C01817=1103.978,373.015,410.367,-179.779,17.252,151.645
C01818=1103.984,373.262,410.332,-179.776,17.255,151.645
C01819=1103.989,373.509,410.296,-179.773,17.259,151.646
C01820=1103.995,373.757,410.260,-179.770,17.264,151.646
C01821=1104.002,374.004,410.224,-179.768,17.268,151.646
C01822=1104.007,374.251,410.189,-179.765,17.272,151.647
C01823=1104.012,374.499,410.152,-179.762,17.276,151.647
C01824=1104.018,374.745,410.116,-179.760,17.280,151.648
C01825=1104.024,374.993,410.081,-179.757,17.284,151.648
C01826=1104.029,375.240,410.045,-179.754,17.289,151.649
C01827=1104.035,375.487,410.008,-179.751,17.293,151.649
C01828=1104.041,375.735,409.972,-179.748,17.297,151.650
C01829=1104.046,375.982,409.936,-179.746,17.302,151.650
C01830=1104.052,376.229,409.900,-179.743,17.306,151.651
C01831=1104.058,376.476,409.865,-179.740,17.310,151.651
C01832=1104.063,376.724,409.828,-179.737,17.314,151.652
C01833=1104.069,376.971,409.792,-179.735,17.319,151.653
C01834=1104.075,377.218,409.756,-179.732,17.323,151.653
C01835=1104.080,377.466,409.719,-179.728,17.328,151.653
C01836=1104.086,377.713,409.684,-179.727,17.332,151.654
C01837=1104.092,377.960,409.648,-179.724,17.336,151.655
C01838=1104.097,378.208,409.611,-179.721,17.341,151.655
C01839=1104.103,378.454,409.575,-179.718,17.345,151.656
C01840=1104.108,378.702,409.539,-179.716,17.349,151.656
C01841=1104.115,378.949,409.502,-179.713,17.354,151.657
C01842=1104.120,379.195,409.466,-179.710,17.358,151.657
C01843=1104.126,379.443,409.430,-179.707,17.363,151.658
C01844=1104.132,379.690,409.394,-179.704,17.368,151.659
C01845=1104.137,379.938,409.357,-179.702,17.372,151.659
C01846=1104.143,380.185,409.321,-179.699,17.376,151.660
C01847=1104.149,380.432,409.284,-179.696,17.381,151.660
C01848=1104.155,380.680,409.248,-179.694,17.385,151.661
C01849=1104.160,380.927,409.212,-179.691,17.390,151.661
C01850=1104.166,381.174,409.175,-179.689,17.394,151.662
C01851=1104.171,381.422,409.139,-179.686,17.399,151.663
C01852=1104.178,381.669,409.103,-179.683,17.404,151.663
C01853=1104.183,381.915,409.066,-179.680,17.408,151.664
C01854=1104.189,382.162,409.029,-179.678,17.413,151.664
C01855=1104.195,382.410,408.992,-179.674,17.417,151.665
C01856=1104.201,382.657,408.957,-179.673,17.422,151.666
C01857=1104.210,383.071,408.895,-179.668,17.430,151.667
C01858=1104.219,383.485,408.834,-179.663,17.438,151.668
C01859=1104.228,383.899,408.773,-179.659,17.446,151.669
C01860=1104.239,384.314,408.711,-179.655,17.454,151.670
C01861=1104.244,384.561,408.674,-179.652,17.458,151.671
C01862=1104.249,384.808,408.637,-179.649,17.463,151.671
C01863=1104.256,385.055,408.601,-179.647,17.468,151.672
C01864=1104.261,385.302,408.564,-179.644,17.473,151.673
C01865=1104.266,385.549,408.527,-179.641,17.478,151.673
C01866=1104.273,385.796,408.491,-179.639,17.483,151.674
C01867=1104.278,386.043,408.454,-179.636,17.488,151.675
C01868=1104.284,386.291,408.417,-179.634,17.493,151.676
C01869=1104.289,386.537,408.380,-179.631,17.498,151.676
C01870=1104.295,386.785,408.343,-179.629,17.502,151.677
C01871=1104.301,387.032,408.306,-179.626,17.507,151.678
C01872=1104.306,387.279,408.269,-179.624,17.512,151.678
C01873=1104.312,387.526,408.232,-179.621,17.517,151.679
C01874=1104.318,387.773,408.195,-179.619,17.522,151.680
C01875=1104.324,388.020,408.159,-179.616,17.527,151.681
C01876=1104.329,388.267,408.121,-179.613,17.532,151.681
C01877=1104.335,388.514,408.084,-179.611,17.537,151.682
C01878=1104.340,388.762,408.047,-179.609,17.542,151.683
C01879=1104.346,389.009,408.010,-179.606,17.547,151.684
C01880=1104.353,389.256,407.973,-179.603,17.552,151.684
C01881=1104.358,389.503,407.936,-179.601,17.557,151.685
C01882=1104.364,389.750,407.899,-179.598,17.563,151.686
C01883=1104.369,389.996,407.862,-179.596,17.568,151.687
C01884=1104.375,390.244,407.825,-179.593,17.573,151.687
C01885=1104.380,390.491,407.788,-179.591,17.578,151.688
C01886=1104.386,390.738,407.750,-179.588,17.583,151.689
C01887=1104.393,390.985,407.713,-179.586,17.588,151.690
C01888=1104.398,391.232,407.676,-179.583,17.593,151.690
C01889=1104.404,391.479,407.639,-179.581,17.599,151.691
C01890=1104.410,391.726,407.602,-179.578,17.604,151.692
C01891=1104.415,391.974,407.565,-179.576,17.609,151.693
C01892=1104.421,392.220,407.527,-179.573,17.615,151.694
C01893=1104.427,392.468,407.490,-179.570,17.620,151.695
C01894=1104.433,392.715,407.452,-179.568,17.625,151.695
C01895=1104.438,392.962,407.415,-179.565,17.631,151.696
C01896=1104.444,393.209,407.377,-179.563,17.636,151.697
C01897=1104.450,393.456,407.340,-179.561,17.641,151.698
C01898=1104.456,393.703,407.302,-179.558,17.646,151.699
C01899=1104.461,393.950,407.265,-179.556,17.652,151.700
C01900=1104.467,394.197,407.228,-179.553,17.657,151.701
C01901=1104.473,394.444,407.191,-179.551,17.663,151.702
C01902=1104.479,394.691,407.153,-179.549,17.668,151.703
C01903=1104.483,394.939,407.115,-179.547,17.673,151.703
C01904=1104.489,395.185,407.077,-179.544,17.679,151.704
C01905=1104.495,395.432,407.040,-179.541,17.685,151.705
C01906=1104.501,395.680,407.003,-179.539,17.690,151.706
C01907=1104.507,395.926,406.965,-179.537,17.696,151.707
C01908=1104.513,396.173,406.927,-179.534,17.701,151.708
C01909=1104.518,396.387,406.895,-179.533,17.706,151.709
C01910=1104.523,396.600,406.862,-179.530,17.711,151.709
C01911=1104.528,396.813,406.830,-179.529,17.716,151.710
C01912=1104.533,397.026,406.797,-179.526,17.721,151.711
C01913=1104.537,397.239,406.764,-179.524,17.725,151.712
C01914=1104.542,397.453,406.731,-179.522,17.731,151.713
C01915=1104.547,397.666,406.699,-179.520,17.735,151.714
C01916=1104.552,397.879,406.666,-179.518,17.741,151.714
C01917=1104.557,398.126,406.629,-179.516,17.746,151.715
C01918=1104.563,398.373,406.592,-179.513,17.752,151.716
C01919=1104.569,398.621,406.553,-179.511,17.757,151.717
C01920=1104.575,398.868,406.515,-179.509,17.763,151.718
C01921=1104.581,399.114,406.477,-179.506,17.769,151.719
C01922=1104.586,399.361,406.440,-179.504,17.775,151.720
C01923=1104.592,399.608,406.401,-179.502,17.781,151.721
C01924=1104.597,399.855,406.364,-179.500,17.786,151.722
C01925=1104.604,400.103,406.326,-179.497,17.793,151.723
C01926=1104.609,400.350,406.288,-179.495,17.798,151.724
C01927=1104.615,400.597,406.250,-179.493,17.804,151.725
C01928=1104.620,400.844,406.212,-179.491,17.810,151.727
C01929=1104.626,401.090,406.174,-179.488,17.816,151.728
C01930=1104.631,401.338,406.136,-179.486,17.822,151.729
C01931=1104.638,401.585,406.098,-179.484,17.828,151.730
C01932=1104.643,401.832,406.060,-179.482,17.834,151.731
C01933=1104.649,402.079,406.021,-179.479,17.840,151.732
C01934=1104.655,402.326,405.984,-179.477,17.846,151.733
C01935=1104.660,402.573,405.945,-179.475,17.852,151.734
C01936=1104.666,402.820,405.907,-179.472,17.859,151.735
C01937=1104.671,403.067,405.869,-179.470,17.865,151.736
C01938=1104.678,403.313,405.830,-179.468,17.871,151.737
C01939=1104.683,403.560,405.792,-179.465,17.877,151.738
C01940=1104.689,403.808,405.754,-179.463,17.883,151.739
C01941=1104.694,404.055,405.716,-179.462,17.889,151.741
C01942=1104.700,404.302,405.678,-179.459,17.896,151.742
C01943=1104.706,404.549,405.639,-179.457,17.902,151.743
C01944=1104.712,404.796,405.600,-179.455,17.908,151.744
C01945=1104.717,405.042,405.562,-179.453,17.915,151.745
C01946=1104.723,405.290,405.524,-179.451,17.921,151.746
C01947=1104.729,405.537,405.486,-179.448,17.928,151.748
C01948=1104.735,405.783,405.447,-179.446,17.933,151.749
C01949=1104.740,406.030,405.408,-179.444,17.940,151.750
C01950=1104.746,406.277,405.371,-179.442,17.946,151.751
C01951=1104.752,406.524,405.331,-179.440,17.953,151.752
C01952=1104.757,406.771,405.293,-179.437,17.960,151.754
C01953=1104.763,407.018,405.255,-179.435,17.965,151.755
C01954=1104.769,407.265,405.216,-179.433,17.972,151.756
C01955=1104.774,407.512,405.177,-179.431,17.979,151.757
C01956=1104.780,407.758,405.139,-179.429,17.986,151.758
C01957=1104.786,408.006,405.100,-179.427,17.992,151.760
C01958=1104.791,408.253,405.062,-179.424,17.999,151.761
C01959=1104.797,408.500,405.023,-179.423,18.005,151.762
C01960=1104.802,408.747,404.984,-179.420,18.012,151.763
C01961=1104.809,408.994,404.945,-179.418,18.018,151.765
C01962=1104.814,409.241,404.907,-179.416,18.026,151.766
C01963=1104.820,409.488,404.868,-179.414,18.032,151.767
C01964=1104.825,409.735,404.829,-179.412,18.039,151.769
C01965=1104.830,409.948,404.795,-179.410,18.045,151.770
C01966=1104.835,410.161,404.762,-179.408,18.051,151.771
C01967=1104.840,410.374,404.728,-179.407,18.056,151.772
C01968=1104.845,410.587,404.696,-179.405,18.062,151.773
C01969=1104.849,410.800,404.662,-179.403,18.068,151.774
C01970=1104.854,411.013,404.628,-179.401,18.074,151.775
C01971=1104.860,411.226,404.595,-179.399,18.080,151.776
C01972=1104.864,411.439,404.561,-179.398,18.086,151.778
C01973=1104.869,411.686,404.522,-179.395,18.093,151.779
C01974=1104.876,411.933,404.483,-179.393,18.100,151.780
C01975=1104.882,412.179,404.444,-179.392,18.107,151.782
C01976=1104.888,412.426,404.405,-179.389,18.114,151.783
C01977=1104.893,412.673,404.367,-179.387,18.121,151.784
C01978=1104.899,412.921,404.327,-179.385,18.128,151.786
C01979=1104.905,413.167,404.288,-179.383,18.135,151.787
C01980=1104.911,413.414,404.249,-179.381,18.142,151.789
C01981=1104.916,413.661,404.210,-179.379,18.149,151.790
C01982=1104.922,413.908,404.171,-179.377,18.156,151.791
C01983=1104.927,414.155,404.132,-179.375,18.164,151.793
C01984=1104.933,414.402,404.092,-179.374,18.171,151.794
C01985=1104.939,414.648,404.053,-179.371,18.178,151.796
C01986=1104.945,414.896,404.014,-179.369,18.185,151.797
C01987=1104.950,415.142,403.975,-179.367,18.193,151.799
C01988=1104.956,415.389,403.935,-179.365,18.200,151.800
C01989=1104.962,415.636,403.896,-179.363,18.207,151.802
C01990=1104.968,415.883,403.857,-179.361,18.215,151.803
C01991=1104.973,416.129,403.818,-179.359,18.222,151.804
C01992=1104.980,416.376,403.778,-179.358,18.229,151.806
C01993=1104.985,416.623,403.739,-179.355,18.236,151.807
C01994=1104.991,416.870,403.700,-179.353,18.244,151.809
C01995=1104.996,417.117,403.660,-179.351,18.252,151.810
C01996=1105.002,417.364,403.621,-179.349,18.259,151.812
C01997=1105.007,417.610,403.582,-179.348,18.267,151.814
C01998=1105.014,417.857,403.542,-179.346,18.274,151.815
C01999=1105.019,418.103,403.502,-179.344,18.282,151.817
C02000=1105.025,418.351,403.462,-179.342,18.290,151.818
C02001=1105.031,418.598,403.423,-179.340,18.297,151.820
C02002=1105.036,418.844,403.384,-179.338,18.305,151.821
C02003=1105.042,419.091,403.344,-179.336,18.313,151.823
C02004=1105.047,419.337,403.304,-179.334,18.321,151.825
C02005=1105.053,419.584,403.265,-179.333,18.328,151.826
C02006=1105.059,419.831,403.226,-179.331,18.336,151.828
C02007=1105.065,420.077,403.185,-179.329,18.344,151.830
C02008=1105.071,420.325,403.145,-179.327,18.352,151.831
C02009=1105.076,420.571,403.106,-179.325,18.360,151.833
C02010=1105.082,420.818,403.066,-179.323,18.368,151.834
C02011=1105.087,421.065,403.027,-179.321,18.375,151.836
C02012=1105.093,421.312,402.987,-179.319,18.383,151.838
C02013=1105.100,421.558,402.947,-179.318,18.392,151.839
C02014=1105.104,421.805,402.907,-179.316,18.400,151.841
C02015=1105.111,422.051,402.867,-179.314,18.408,151.843
C02016=1105.117,422.299,402.828,-179.312,18.416,151.844
C02017=1105.122,422.545,402.787,-179.310,18.424,151.846
C02018=1105.128,422.792,402.748,-179.308,18.432,151.848
C02019=1105.134,423.038,402.708,-179.307,18.440,151.850
C02020=1105.139,423.285,402.668,-179.305,18.448,151.851
C02021=1105.144,423.505,402.632,-179.304,18.455,151.853
C02022=1105.150,423.724,402.597,-179.302,18.463,151.854
C02023=1105.155,423.944,402.561,-179.300,18.470,151.856
C02024=1105.160,424.164,402.526,-179.299,18.477,151.858
C02025=1105.164,424.383,402.490,-179.297,18.485,151.859
C02026=1105.169,424.604,402.454,-179.296,18.492,151.861
C02027=1105.174,424.822,402.418,-179.294,18.500,151.862
C02028=1105.179,425.043,402.382,-179.293,18.507,151.864
C02029=1105.186,425.289,402.342,-179.291,18.516,151.866
C02030=1105.191,425.536,402.303,-179.290,18.524,151.868
C02031=1105.197,425.782,402.262,-179.288,18.533,151.869
C02032=1105.203,426.029,402.222,-179.286,18.542,151.871
C02033=1105.208,426.275,402.182,-179.284,18.550,151.873
C02034=1105.214,426.523,402.142,-179.282,18.559,151.875
C02035=1105.220,426.769,402.102,-179.281,18.567,151.877
C02036=1105.226,427.016,402.061,-179.279,18.576,151.879
C02037=1105.231,427.262,402.021,-179.278,18.584,151.881
C02038=1105.237,427.509,401.980,-179.277,18.593,151.883
C02039=1105.243,427.755,401.940,-179.274,18.602,151.885
C02040=1105.249,428.002,401.900,-179.273,18.611,151.886
C02041=1105.254,428.249,401.860,-179.271,18.619,151.888
C02042=1105.260,428.495,401.819,-179.270,18.628,151.890
C02043=1105.266,428.742,401.779,-179.268,18.637,151.892
C02044=1105.272,428.989,401.738,-179.266,18.646,151.894
C02045=1105.277,429.236,401.698,-179.265,18.655,151.896
C02046=1105.283,429.481,401.658,-179.263,18.664,151.898
C02047=1105.289,429.728,401.617,-179.262,18.673,151.900
C02048=1105.294,429.975,401.576,-179.260,18.682,151.902
C02049=1105.300,430.221,401.535,-179.259,18.691,151.904
C02050=1105.306,430.467,401.495,-179.257,18.700,151.906
C02051=1105.312,430.714,401.454,-179.255,18.710,151.908
C02052=1105.317,430.961,401.414,-179.254,18.719,151.910
C02053=1105.323,431.208,401.373,-179.253,18.728,151.912
C02054=1105.329,431.454,401.332,-179.251,18.737,151.914
C02055=1105.334,431.700,401.292,-179.249,18.747,151.917
C02056=1105.340,431.946,401.251,-179.248,18.756,151.919
C02057=1105.346,432.193,401.210,-179.247,18.765,151.921
C02058=1105.352,432.440,401.169,-179.245,18.775,151.923
C02059=1105.357,432.687,401.129,-179.244,18.784,151.925
C02060=1105.363,432.933,401.087,-179.243,18.793,151.927
C02061=1105.368,433.179,401.047,-179.241,18.803,151.929
C02062=1105.375,433.426,401.007,-179.240,18.812,151.931
C02063=1105.381,433.672,400.965,-179.238,18.822,151.934
C02064=1105.386,433.919,400.924,-179.237,18.832,151.936
C02065=1105.392,434.166,400.884,-179.236,18.841,151.938
C02066=1105.398,434.412,400.842,-179.234,18.851,151.940
C02067=1105.403,434.659,400.802,-179.233,18.861,151.943
C02068=1105.408,434.904,400.760,-179.231,18.870,151.945
C02069=1105.414,435.151,400.719,-179.230,18.880,151.947
C02070=1105.419,435.398,400.678,-179.229,18.890,151.949
C02071=1105.425,435.644,400.637,-179.228,18.900,151.951
C02072=1105.431,435.891,400.596,-179.226,18.910,151.954
C02073=1105.437,436.137,400.555,-179.225,18.919,151.956
C02074=1105.443,436.384,400.513,-179.224,18.930,151.958
C02075=1105.448,436.630,400.472,-179.223,18.940,151.961
C02076=1105.454,436.877,400.431,-179.221,18.950,151.963
C02077=1105.459,437.090,400.395,-179.220,18.958,151.965
C02078=1105.464,437.303,400.360,-179.219,18.967,151.967
C02079=1105.468,437.516,400.324,-179.219,18.976,151.969
C02080=1105.474,437.731,400.288,-179.217,18.985,151.971
C02081=1105.479,437.944,400.253,-179.216,18.994,151.973
C02082=1105.484,438.157,400.216,-179.215,19.002,151.975
C02083=1105.489,438.371,400.181,-179.214,19.011,151.977
C02084=1105.494,438.584,400.145,-179.213,19.020,151.979
C02085=1105.500,438.831,400.104,-179.212,19.030,151.982
C02086=1105.506,439.077,400.063,-179.210,19.041,151.984
C02087=1105.511,439.324,400.021,-179.209,19.052,151.987
C02088=1105.517,439.570,399.980,-179.208,19.062,151.989
C02089=1105.523,439.816,399.938,-179.207,19.072,151.992
C02090=1105.529,440.062,399.897,-179.206,19.083,151.994
C02091=1105.535,440.309,399.855,-179.205,19.093,151.997
C02092=1105.539,440.556,399.814,-179.204,19.104,151.999
C02093=1105.545,440.802,399.772,-179.203,19.114,152.002
C02094=1105.551,441.048,399.731,-179.202,19.125,152.004
C02095=1105.557,441.294,399.689,-179.200,19.136,152.007
C02096=1105.562,441.541,399.647,-179.200,19.147,152.009
C02097=1105.568,441.787,399.606,-179.199,19.158,152.012
C02098=1105.574,442.033,399.564,-179.197,19.169,152.014
C02099=1105.580,442.280,399.522,-179.197,19.179,152.017
C02100=1105.586,442.526,399.481,-179.196,19.190,152.020
C02101=1105.591,442.772,399.439,-179.195,19.202,152.022
C02102=1105.597,443.018,399.397,-179.194,19.212,152.025
C02103=1105.603,443.264,399.355,-179.193,19.223,152.028
C02104=1105.608,443.511,399.313,-179.192,19.235,152.030
C02105=1105.614,443.757,399.272,-179.191,19.245,152.033
C02106=1105.620,444.004,399.229,-179.190,19.257,152.036
C02107=1105.626,444.250,399.188,-179.190,19.268,152.039
C02108=1105.631,444.497,399.146,-179.190,19.278,152.041
C02109=1105.637,444.743,399.104,-179.190,19.290,152.044
C02110=1105.643,444.989,399.062,-179.190,19.301,152.047
C02111=1105.648,445.235,399.020,-179.190,19.312,152.050
C02112=1105.654,445.482,398.978,-179.190,19.323,152.053
C02113=1105.660,445.727,398.936,-179.190,19.333,152.055
C02114=1105.666,445.975,398.894,-179.190,19.345,152.058
C02115=1105.672,446.221,398.852,-179.191,19.355,152.061
C02116=1105.677,446.467,398.810,-179.192,19.366,152.064
C02117=1105.683,446.713,398.768,-179.192,19.377,152.067
C02118=1105.688,446.959,398.726,-179.193,19.388,152.070
C02119=1105.694,447.206,398.684,-179.194,19.399,152.073
C02120=1105.700,447.452,398.642,-179.195,19.410,152.076
C02121=1105.706,447.699,398.599,-179.197,19.421,152.079
C02122=1105.711,447.945,398.557,-179.198,19.432,152.082
C02123=1105.717,448.191,398.515,-179.199,19.443,152.085
C02124=1105.722,448.437,398.473,-179.201,19.453,152.088
C02125=1105.728,448.683,398.430,-179.201,19.464,152.091
C02126=1105.734,448.930,398.388,-179.203,19.475,152.094
C02127=1105.740,449.177,398.346,-179.205,19.486,152.097
C02128=1105.745,449.423,398.303,-179.207,19.496,152.100
C02129=1105.751,449.669,398.262,-179.209,19.507,152.103
C02130=1105.757,449.915,398.219,-179.211,19.517,152.106
C02131=1105.762,450.162,398.177,-179.213,19.529,152.109
C02132=1105.769,450.407,398.135,-179.215,19.539,152.112
C02133=1105.364,450.401,398.011,-179.292,19.769,152.185
C02134=1105.357,450.155,398.053,-179.290,19.758,152.182
C02135=1105.352,449.909,398.095,-179.288,19.747,152.179
C02136=1105.346,449.662,398.138,-179.286,19.736,152.175
C02137=1105.340,449.416,398.180,-179.284,19.726,152.172
C02138=1105.335,449.170,398.222,-179.283,19.715,152.169
C02139=1105.329,448.924,398.265,-179.282,19.704,152.166
C02140=1105.323,448.678,398.307,-179.280,19.693,152.163
C02141=1105.317,448.431,398.349,-179.278,19.682,152.160
C02142=1105.312,448.185,398.392,-179.277,19.671,152.157
C02143=1105.307,447.938,398.434,-179.275,19.661,152.154
C02144=1105.301,447.692,398.475,-179.274,19.649,152.151
C02145=1105.294,447.446,398.519,-179.273,19.638,152.148
C02146=1105.289,447.199,398.561,-179.273,19.627,152.145
C02147=1105.283,446.953,398.603,-179.272,19.616,152.142
C02148=1105.278,446.707,398.645,-179.271,19.605,152.139
C02149=1105.273,446.460,398.687,-179.270,19.594,152.136
C02150=1105.266,446.215,398.729,-179.269,19.583,152.133
C02151=1105.260,445.968,398.771,-179.269,19.572,152.130
C02152=1105.255,445.721,398.813,-179.268,19.561,152.127
C02153=1105.249,445.476,398.856,-179.269,19.550,152.125
C02154=1105.243,445.229,398.897,-179.268,19.539,152.122
C02155=1105.238,444.983,398.939,-179.268,19.528,152.119
C02156=1105.231,444.737,398.982,-179.268,19.517,152.116
C02157=1105.226,444.490,399.024,-179.268,19.506,152.113
C02158=1105.220,444.244,399.065,-179.269,19.495,152.111
C02159=1105.215,443.997,399.107,-179.270,19.483,152.108
C02160=1105.208,443.752,399.149,-179.270,19.473,152.105
C02161=1105.203,443.505,399.192,-179.271,19.461,152.102
C02162=1105.197,443.259,399.233,-179.272,19.450,152.100
C02163=1105.192,443.013,399.275,-179.273,19.439,152.097
C02164=1105.186,442.766,399.316,-179.274,19.428,152.094
C02165=1105.181,442.520,399.359,-179.274,19.417,152.092
C02166=1105.174,442.274,399.401,-179.276,19.406,152.089
C02167=1105.168,442.027,399.443,-179.277,19.395,152.086
C02168=1105.163,441.781,399.485,-179.278,19.383,152.084
C02169=1105.157,441.535,399.526,-179.279,19.373,152.081
C02170=1105.151,441.288,399.567,-179.280,19.362,152.079
C02171=1105.146,441.042,399.610,-179.281,19.351,152.076
C02172=1105.140,440.796,399.651,-179.282,19.340,152.074
C02173=1105.134,440.549,399.692,-179.283,19.329,152.071
C02174=1105.129,440.303,399.735,-179.285,19.319,152.068
C02175=1105.123,440.057,399.776,-179.286,19.309,152.066
C02176=1105.117,439.811,399.817,-179.287,19.298,152.064
C02177=1105.111,439.564,399.859,-179.288,19.287,152.061
C02178=1105.105,439.318,399.900,-179.289,19.277,152.059
C02179=1105.100,439.071,399.942,-179.291,19.266,152.056
C02180=1105.094,438.825,399.983,-179.291,19.256,152.054
C02181=1105.088,438.579,400.025,-179.293,19.245,152.051
C02182=1105.083,438.367,400.060,-179.294,19.236,152.049
C02183=1105.078,438.156,400.096,-179.295,19.228,152.047
C02184=1105.073,437.945,400.131,-179.296,19.218,152.045
C02185=1105.068,437.733,400.167,-179.297,19.210,152.043
C02186=1105.063,437.522,400.202,-179.298,19.201,152.041
C02187=1105.058,437.311,400.237,-179.300,19.192,152.039
C02188=1105.054,437.100,400.272,-179.300,19.184,152.037
C02189=1105.048,436.889,400.309,-179.302,19.175,152.035
C02190=1105.042,436.642,400.349,-179.303,19.165,152.033
C02191=1105.037,436.396,400.390,-179.304,19.154,152.030
C02192=1105.031,436.149,400.431,-179.305,19.145,152.028
C02193=1105.025,435.903,400.473,-179.307,19.134,152.026
C02194=1105.017,435.527,400.536,-179.309,19.119,152.022
C02195=1105.008,435.152,400.598,-179.311,19.104,152.019
C02196=1104.999,434.776,400.662,-179.313,19.089,152.015
C02197=1104.991,434.401,400.724,-179.315,19.074,152.012
C02198=1104.985,434.154,400.765,-179.317,19.064,152.009
C02199=1104.979,433.908,400.805,-179.318,19.055,152.007
C02200=1104.974,433.662,400.846,-179.320,19.045,152.005
C02201=1104.968,433.415,400.887,-179.321,19.035,152.003
C02202=1104.962,433.169,400.929,-179.322,19.026,152.001
C02203=1104.957,432.922,400.969,-179.324,19.016,151.999
C02204=1104.951,432.675,401.010,-179.325,19.007,151.996
C02205=1104.944,432.430,401.051,-179.327,18.997,151.994
C02206=1104.939,432.183,401.092,-179.328,18.988,151.992
C02207=1104.933,431.936,401.133,-179.329,18.978,151.990
C02208=1104.928,431.690,401.173,-179.332,18.969,151.988
C02209=1104.922,431.444,401.214,-179.333,18.959,151.986
C02210=1104.917,431.197,401.255,-179.334,18.950,151.984
C02211=1104.911,430.950,401.296,-179.336,18.941,151.982
C02212=1104.905,430.703,401.336,-179.337,18.932,151.980
C02213=1104.899,430.457,401.376,-179.339,18.922,151.978
C02214=1104.894,430.211,401.418,-179.340,18.914,151.976
C02215=1104.888,429.964,401.459,-179.342,18.904,151.973
C02216=1104.882,429.717,401.499,-179.344,18.895,151.971
C02217=1104.876,429.471,401.539,-179.345,18.886,151.970
C02218=1104.871,429.225,401.580,-179.347,18.876,151.967
C02219=1104.865,428.978,401.621,-179.348,18.868,151.965
C02220=1104.859,428.731,401.661,-179.350,18.859,151.963
C02221=1104.853,428.485,401.701,-179.351,18.850,151.961
C02222=1104.848,428.238,401.742,-179.353,18.841,151.960
C02223=1104.841,427.991,401.782,-179.355,18.832,151.958
C02224=1104.836,427.745,401.823,-179.357,18.823,151.956
C02225=1104.830,427.498,401.863,-179.358,18.814,151.954
C02226=1104.824,427.252,401.904,-179.360,18.806,151.952
C02227=1104.818,427.005,401.944,-179.361,18.797,151.950
C02228=1104.813,426.759,401.984,-179.364,18.788,151.948
C02229=1104.807,426.512,402.024,-179.365,18.779,151.946
C02230=1104.802,426.265,402.065,-179.367,18.771,151.944
C02231=1104.795,426.018,402.105,-179.368,18.762,151.942
C02232=1104.790,425.772,402.145,-179.370,18.754,151.941
C02233=1104.784,425.526,402.186,-179.372,18.745,151.939
C02234=1104.779,425.278,402.226,-179.374,18.736,151.937
C02235=1104.773,425.031,402.266,-179.376,18.728,151.935
C02236=1104.767,424.786,402.306,-179.377,18.719,151.933
C02237=1104.761,424.539,402.347,-179.379,18.711,151.931
C02238=1104.754,424.228,402.397,-179.381,18.700,151.929
C02239=1104.747,423.917,402.447,-179.383,18.690,151.927
C02240=1104.740,423.607,402.498,-179.386,18.679,151.925
C02241=1104.733,423.296,402.548,-179.387,18.669,151.922
C02242=1104.727,423.050,402.588,-179.389,18.661,151.921
C02243=1104.721,422.802,402.628,-179.392,18.652,151.919
C02244=1104.715,422.556,402.668,-179.393,18.644,151.917
C02245=1104.710,422.309,402.708,-179.395,18.636,151.915
C02246=1104.704,422.063,402.748,-179.397,18.627,151.914
C02247=1104.698,421.816,402.788,-179.399,18.619,151.912
C02248=1104.693,421.569,402.828,-179.401,18.611,151.910
C02249=1104.687,421.322,402.867,-179.403,18.603,151.909
C02250=1104.680,421.076,402.908,-179.404,18.596,151.907
C02251=1104.676,420.829,402.947,-179.406,18.588,151.905
C02252=1104.670,420.582,402.987,-179.408,18.580,151.904
C02253=1104.664,420.336,403.026,-179.410,18.572,151.902
C02254=1104.658,420.089,403.066,-179.411,18.564,151.900
C02255=1104.652,419.842,403.107,-179.414,18.556,151.899
C02256=1104.647,419.596,403.146,-179.415,18.548,151.897
C02257=1104.641,419.349,403.185,-179.417,18.540,151.895
C02258=1104.636,419.102,403.225,-179.419,18.532,151.894
C02259=1104.629,418.855,403.265,-179.421,18.524,151.892
C02260=1104.623,418.608,403.304,-179.423,18.517,151.891
C02261=1104.618,418.362,403.343,-179.425,18.508,151.889
C02262=1104.613,418.114,403.383,-179.427,18.501,151.887
C02263=1104.607,417.869,403.423,-179.429,18.494,151.886
C02264=1104.601,417.621,403.463,-179.431,18.486,151.884
C02265=1104.595,417.375,403.502,-179.433,18.478,151.883
C02266=1104.589,417.128,403.541,-179.435,18.470,151.881
C02267=1104.584,416.881,403.581,-179.437,18.463,151.880
C02268=1104.578,416.634,403.620,-179.439,18.455,151.878
C02269=1104.572,416.387,403.660,-179.440,18.448,151.877
C02270=1104.567,416.140,403.699,-179.443,18.441,151.875
C02271=1104.561,415.893,403.738,-179.445,18.433,151.874
C02272=1104.555,415.647,403.778,-179.447,18.425,151.872
C02273=1104.549,415.400,403.817,-179.448,18.419,151.871
C02274=1104.543,415.154,403.856,-179.451,18.411,151.869
C02275=1104.537,414.907,403.896,-179.453,18.404,151.868
C02276=1104.532,414.660,403.934,-179.455,18.396,151.866
C02277=1104.526,414.412,403.974,-179.457,18.389,151.865
C02278=1104.521,414.166,404.013,-179.459,18.382,151.863
C02279=1104.515,413.919,404.052,-179.461,18.374,151.862
C02280=1104.509,413.672,404.091,-179.463,18.367,151.861
C02281=1104.503,413.425,404.131,-179.465,18.360,151.859
C02282=1104.498,413.179,404.170,-179.467,18.353,151.858
C02283=1104.491,412.932,404.209,-179.469,18.345,151.856
C02284=1104.486,412.685,404.247,-179.471,18.339,151.855
C02285=1104.480,412.438,404.287,-179.473,18.331,151.854
C02286=1104.475,412.191,404.326,-179.476,18.324,151.852
C02287=1104.469,411.944,404.365,-179.477,18.318,151.851
C02288=1104.463,411.698,404.404,-179.479,18.310,151.849
C02289=1104.457,411.450,404.443,-179.482,18.303,151.848
C02290=1104.452,411.237,404.477,-179.483,18.298,151.847
C02291=1104.447,411.024,404.510,-179.485,18.291,151.846
C02292=1104.442,410.811,404.544,-179.487,18.285,151.845
C02293=1104.437,410.597,404.577,-179.489,18.279,151.843
C02294=1104.433,410.384,404.611,-179.491,18.273,151.842
C02295=1104.428,410.171,404.645,-179.493,18.267,151.841
C02296=1104.423,409.957,404.678,-179.495,18.261,151.840
C02297=1104.418,409.744,404.712,-179.496,18.256,151.839
C02298=1104.412,409.498,404.751,-179.498,18.249,151.838
C02299=1104.407,409.250,404.789,-179.500,18.242,151.836
C02300=1104.401,409.004,404.828,-179.502,18.235,151.835
C02301=1104.396,408.757,404.867,-179.505,18.228,151.834
C02302=1104.389,408.510,404.906,-179.507,18.222,151.832
C02303=1104.384,408.263,404.944,-179.509,18.215,151.831
C02304=1104.379,408.016,404.983,-179.511,18.208,151.830
C02305=1104.373,407.769,405.022,-179.513,18.201,151.829
C02306=1104.367,407.522,405.060,-179.515,18.195,151.827
C02307=1104.361,407.275,405.099,-179.518,18.188,151.826
C02308=1104.355,407.028,405.138,-179.520,18.182,151.825
C02309=1104.350,406.781,405.176,-179.522,18.175,151.824
C02310=1104.344,406.534,405.214,-179.524,18.169,151.822
C02311=1104.338,406.287,405.254,-179.527,18.162,151.821
C02312=1104.333,406.040,405.292,-179.528,18.155,151.820
C02313=1104.327,405.794,405.330,-179.530,18.150,151.819
C02314=1104.321,405.546,405.369,-179.533,18.143,151.818
C02315=1104.316,405.299,405.407,-179.535,18.136,151.816
C02316=1104.310,405.053,405.445,-179.538,18.130,151.815
C02317=1104.304,404.805,405.485,-179.539,18.123,151.814
C02318=1104.298,404.559,405.522,-179.542,18.117,151.813
C02319=1104.293,404.312,405.561,-179.544,18.111,151.812
C02320=1104.287,404.065,405.599,-179.546,18.105,151.811
C02321=1104.281,403.817,405.637,-179.549,18.098,151.810
C02322=1104.276,403.571,405.676,-179.551,18.092,151.808
C02323=1104.270,403.324,405.714,-179.553,18.086,151.807
C02324=1104.264,403.076,405.753,-179.555,18.080,151.806
C02325=1104.258,402.829,405.791,-179.557,18.074,151.805
C02326=1104.253,402.582,405.829,-179.559,18.068,151.804
C02327=1104.247,402.336,405.867,-179.562,18.061,151.803
C02328=1104.242,402.089,405.905,-179.564,18.055,151.802
C02329=1104.235,401.841,405.943,-179.566,18.049,151.801
C02330=1104.230,401.594,405.981,-179.569,18.042,151.799
C02331=1104.224,401.347,406.019,-179.571,18.037,151.798
C02332=1104.218,401.101,406.057,-179.573,18.031,151.797
C02333=1104.213,400.854,406.095,-179.576,18.025,151.796
C02334=1104.207,400.606,406.133,-179.578,18.019,151.795
C02335=1104.202,400.359,406.172,-179.580,18.013,151.794
C02336=1104.196,400.112,406.210,-179.582,18.007,151.793
C02337=1104.190,399.866,406.247,-179.585,18.000,151.792
C02338=1104.185,399.619,406.286,-179.587,17.995,151.791
C02339=1104.178,399.371,406.324,-179.589,17.989,151.790
C02340=1104.172,399.124,406.362,-179.591,17.983,151.789
C02341=1104.167,398.877,406.400,-179.594,17.977,151.788
C02342=1104.161,398.631,406.438,-179.597,17.971,151.787
C02343=1104.155,398.384,406.475,-179.599,17.965,151.786
C02344=1104.150,398.136,406.513,-179.601,17.960,151.785
C02345=1104.144,397.889,406.551,-179.603,17.954,151.784
C02346=1104.139,397.676,406.583,-179.605,17.949,151.783
C02347=1104.134,397.462,406.616,-179.607,17.944,151.782
C02348=1104.129,397.249,406.649,-179.609,17.939,151.781
C02349=1104.124,397.036,406.681,-179.611,17.934,151.781
C02350=1104.120,396.822,406.714,-179.614,17.929,151.780
C02351=1104.115,396.609,406.747,-179.615,17.924,151.779
C02352=1104.110,396.396,406.780,-179.618,17.919,151.778
C02353=1104.105,396.183,406.812,-179.620,17.915,151.777
C02354=1104.099,395.935,406.850,-179.622,17.909,151.776
C02355=1104.093,395.688,406.887,-179.625,17.903,151.775
C02356=1104.087,395.441,406.925,-179.627,17.897,151.775
C02357=1104.082,395.194,406.963,-179.629,17.892,151.774
C02358=1104.076,394.947,407.000,-179.632,17.886,151.773
C02359=1104.070,394.700,407.038,-179.634,17.881,151.772
C02360=1104.065,394.453,407.075,-179.636,17.875,151.771
C02361=1104.059,394.206,407.113,-179.639,17.870,151.770
C02362=1104.053,393.959,407.150,-179.641,17.865,151.769
C02363=1104.047,393.712,407.187,-179.643,17.859,151.768
C02364=1104.041,393.465,407.225,-179.647,17.853,151.767
C02365=1104.036,393.218,407.262,-179.649,17.848,151.766
C02366=1104.030,392.971,407.300,-179.651,17.842,151.766
C02367=1104.025,392.723,407.338,-179.654,17.837,151.765
C02368=1104.019,392.477,407.375,-179.656,17.832,151.764
C02369=1104.014,392.229,407.412,-179.659,17.827,151.763
C02370=1104.007,391.982,407.449,-179.661,17.821,151.762
C02371=1104.001,391.735,407.487,-179.663,17.816,151.761
C02372=1103.996,391.488,407.524,-179.666,17.811,151.761
C02373=1103.990,391.241,407.561,-179.668,17.806,151.760
C02374=1103.984,390.994,407.598,-179.671,17.801,151.759
C02375=1103.979,390.747,407.636,-179.673,17.795,151.758
C02376=1103.973,390.500,407.673,-179.676,17.790,151.757
C02377=1103.967,390.252,407.710,-179.678,17.785,151.756
C02378=1103.962,390.005,407.747,-179.681,17.780,151.756
C02379=1103.955,389.759,407.785,-179.683,17.774,151.755
C02380=1103.950,389.512,407.821,-179.686,17.769,151.754
C02381=1103.944,389.265,407.858,-179.688,17.764,151.753
C02382=1103.938,389.018,407.896,-179.691,17.759,151.753
C02383=1103.933,388.771,407.933,-179.693,17.754,151.752
C02384=1103.927,388.523,407.970,-179.696,17.749,151.751
C02385=1103.921,388.276,408.007,-179.699,17.743,151.750
C02386=1103.915,388.029,408.044,-179.702,17.738,151.750
C02387=1103.909,387.782,408.081,-179.704,17.734,151.749
C02388=1103.904,387.535,408.118,-179.706,17.729,151.748
C02389=1103.899,387.288,408.155,-179.709,17.723,151.747
C02390=1103.892,387.041,408.191,-179.712,17.719,151.747
C02391=1103.887,386.794,408.229,-179.714,17.714,151.746
C02392=1103.881,386.546,408.266,-179.717,17.708,151.745
C02393=1103.876,386.299,408.303,-179.719,17.704,151.744
C02394=1103.870,386.052,408.339,-179.722,17.699,151.744
C02395=1103.864,385.805,408.376,-179.724,17.693,151.743
C02396=1103.859,385.558,408.413,-179.727,17.689,151.742
C02397=1103.853,385.311,408.450,-179.730,17.684,151.741
C02398=1103.847,385.064,408.487,-179.733,17.679,151.741
C02399=1103.842,384.817,408.523,-179.735,17.674,151.740
C02400=1103.836,384.569,408.560,-179.738,17.669,151.739
C02401=1103.831,384.322,408.597,-179.740,17.664,151.739
C02402=1103.821,383.908,408.658,-179.745,17.656,151.738
C02403=1103.812,383.493,408.720,-179.749,17.648,151.736
C02404=1103.802,383.079,408.782,-179.754,17.640,151.735
C02405=1103.792,382.665,408.843,-179.758,17.632,151.734
C02406=1103.786,382.417,408.880,-179.761,17.627,151.734
C02407=1103.781,382.170,408.915,-179.764,17.622,151.733
C02408=1103.775,381.923,408.952,-179.766,17.618,151.732
C02409=1103.769,381.676,408.989,-179.769,17.613,151.732
C02410=1103.763,381.429,409.026,-179.771,17.609,151.731
C02411=1103.758,381.182,409.061,-179.774,17.604,151.730
C02412=1103.752,380.934,409.098,-179.777,17.599,151.730
C02413=1103.746,380.687,409.135,-179.780,17.594,151.729
C02414=1103.740,380.440,409.172,-179.782,17.590,151.729
C02415=1103.735,380.193,409.207,-179.785,17.586,151.728
C02416=1103.729,379.945,409.244,-179.788,17.581,151.727
C02417=1103.723,379.698,409.281,-179.790,17.576,151.727
C02418=1103.718,379.451,409.316,-179.793,17.572,151.726
C02419=1103.712,379.204,409.353,-179.796,17.567,151.726
C02420=1103.706,378.956,409.389,-179.798,17.563,151.725
C02421=1103.701,378.710,409.425,-179.801,17.559,151.725
C02422=1103.695,378.463,409.462,-179.804,17.554,151.724
C02423=1103.689,378.215,409.498,-179.807,17.549,151.723
C02424=1103.684,377.968,409.534,-179.810,17.545,151.723
C02425=1103.678,377.721,409.570,-179.812,17.541,151.722
C02426=1103.672,377.473,409.607,-179.815,17.536,151.722
C02427=1103.667,377.226,409.642,-179.818,17.532,151.721
C02428=1103.661,376.979,409.680,-179.821,17.527,151.721
C02429=1103.655,376.731,409.715,-179.823,17.523,151.720
C02430=1103.649,376.484,409.751,-179.826,17.519,151.720
C02431=1103.644,376.237,409.788,-179.829,17.514,151.719
C02432=1103.638,375.990,409.823,-179.832,17.510,151.719
C02433=1103.632,375.743,409.859,-179.834,17.505,151.718
C02434=1103.627,375.495,409.896,-179.837,17.501,151.717
C02435=1103.621,375.248,409.931,-179.840,17.497,151.717
C02436=1103.615,375.001,409.968,-179.843,17.493,151.717
C02437=1103.610,374.754,410.004,-179.846,17.488,151.716
C02438=1103.604,374.506,410.039,-179.848,17.484,151.715
C02439=1103.598,374.259,410.076,-179.851,17.480,151.715
C02440=1103.593,374.012,410.111,-179.854,17.475,151.714
C02441=1103.587,373.764,410.147,-179.856,17.472,151.714
C02442=1103.582,373.517,410.183,-179.859,17.467,151.714
C02443=1103.575,373.270,410.219,-179.862,17.463,151.713
C02444=1103.569,373.022,410.255,-179.865,17.459,151.713
C02445=1103.564,372.775,410.290,-179.868,17.455,151.712
C02446=1103.558,372.528,410.326,-179.871,17.451,151.712
C02447=1103.553,372.281,410.361,-179.874,17.446,151.711
C02448=1103.546,372.034,410.398,-179.876,17.443,151.711
C02449=1103.542,371.786,410.434,-179.879,17.439,151.710
C02450=1103.536,371.539,410.470,-179.882,17.434,151.710
C02451=1103.529,371.291,410.505,-179.885,17.430,151.709
C02452=1103.524,371.044,410.541,-179.888,17.426,151.709
C02453=1103.518,370.796,410.576,-179.891,17.422,151.709
C02454=1103.509,370.409,410.632,-179.895,17.416,151.708
C02455=1103.500,370.021,410.688,-179.899,17.410,151.707
C02456=1103.491,369.633,410.744,-179.904,17.404,151.707
C02457=1103.483,369.246,410.799,-179.909,17.397,151.706
C02458=1103.477,368.999,410.835,-179.911,17.393,151.706
C02459=1103.471,368.752,410.871,-179.914,17.389,151.705
C02460=1103.465,368.504,410.906,-179.917,17.385,151.705
C02461=1103.460,368.257,410.941,-179.920,17.381,151.704
C02462=1103.454,368.009,410.977,-179.923,17.377,151.704
C02463=1103.449,367.762,411.012,-179.926,17.373,151.704
C02464=1103.443,367.514,411.048,-179.929,17.370,151.703
C02465=1103.437,367.267,411.083,-179.932,17.365,151.703
C02466=1103.431,367.020,411.119,-179.934,17.362,151.702
C02467=1103.426,366.773,411.154,-179.937,17.358,151.702
C02468=1103.421,366.525,411.189,-179.940,17.354,151.702
C02469=1103.415,366.277,411.225,-179.943,17.350,151.701
C02470=1103.409,366.030,411.260,-179.946,17.346,151.701
C02471=1103.403,365.783,411.296,-179.949,17.343,151.701
C02472=1103.398,365.535,411.330,-179.952,17.339,151.700
C02473=1103.391,365.288,411.365,-179.955,17.335,151.700
C02474=1103.386,365.041,411.401,-179.958,17.331,151.700
C02475=1103.381,364.793,411.435,-179.961,17.327,151.699
C02476=1103.375,364.546,411.471,-179.964,17.324,151.699
C02477=1103.369,364.299,411.507,-179.967,17.320,151.699
C02478=1103.363,364.051,411.541,-179.969,17.316,151.698
C02479=1103.357,363.804,411.576,-179.973,17.312,151.698
C02480=1103.351,363.556,411.612,-179.975,17.309,151.698
C02481=1103.346,363.308,411.647,-179.978,17.305,151.697
C02482=1103.341,363.061,411.682,-179.982,17.301,151.697
C02483=1103.334,362.813,411.717,-179.984,17.298,151.697
C02484=1103.329,362.566,411.752,-179.988,17.294,151.696
C02485=1103.324,362.319,411.787,-179.990,17.291,151.696
C02486=1103.318,362.071,411.822,-179.994,17.287,151.696
C02487=1103.312,361.824,411.856,-179.996,17.283,151.696
C02488=1103.306,361.576,411.892,-180.000,17.280,151.695
C02489=1103.301,361.329,411.927,179.998,17.276,151.695
C02490=1103.295,361.082,411.961,179.995,17.272,151.695
C02491=1103.289,360.834,411.996,179.992,17.269,151.694
C02492=1103.283,360.587,412.032,179.989,17.265,151.694
C02493=1103.278,360.339,412.066,179.986,17.262,151.694
C02494=1103.272,360.091,412.101,179.983,17.258,151.694
C02495=1103.266,359.844,412.136,179.980,17.255,151.693
C02496=1103.261,359.597,412.170,179.977,17.251,151.693
C02497=1103.255,359.349,412.206,179.974,17.248,151.693
C02498=1103.249,359.102,412.241,179.970,17.244,151.693
C02499=1103.244,358.854,412.275,179.968,17.241,151.692
C02500=1103.238,358.606,412.310,179.965,17.237,151.692
C02501=1103.232,358.359,412.345,179.962,17.234,151.692
C02502=1103.227,358.112,412.379,179.958,17.230,151.692
C02503=1103.221,357.864,412.413,179.956,17.227,151.691
C02504=1103.215,357.616,412.448,179.952,17.223,151.691
C02505=1103.209,357.369,412.483,179.949,17.220,151.691
C02506=1103.200,356.996,412.536,179.945,17.215,151.691
C02507=1103.192,356.624,412.587,179.941,17.210,151.690
C02508=1103.183,356.251,412.639,179.936,17.205,151.690
C02509=1103.175,355.878,412.692,179.931,17.200,151.690
C02510=1103.169,355.631,412.726,179.928,17.197,151.689
C02511=1103.163,355.383,412.761,179.925,17.193,151.689
C02512=1103.158,355.135,412.795,179.922,17.190,151.689
C02513=1103.152,354.888,412.829,179.919,17.187,151.689
C02514=1103.147,354.641,412.863,179.916,17.183,151.689
C02515=1103.142,354.393,412.898,179.913,17.180,151.688
C02516=1103.135,354.145,412.933,179.910,17.176,151.688
C02517=1103.129,353.898,412.967,179.907,17.173,151.688
C02518=1103.124,353.650,413.001,179.903,17.170,151.688
C02519=1103.118,353.403,413.035,179.900,17.167,151.688
C02520=1103.113,353.155,413.070,179.898,17.164,151.688
C02521=1103.107,352.907,413.104,179.894,17.160,151.687
C02522=1103.101,352.660,413.138,179.891,17.157,151.687
C02523=1103.096,352.412,413.173,179.888,17.153,151.687
C02524=1103.090,352.165,413.207,179.885,17.151,151.687
C02525=1103.084,351.917,413.240,179.882,17.148,151.687
C02526=1103.078,351.669,413.275,179.879,17.144,151.687
C02527=1103.073,351.422,413.310,179.876,17.141,151.686
C02528=1103.067,351.174,413.344,179.873,17.138,151.686
C02529=1103.061,350.927,413.378,179.869,17.135,151.686
C02530=1103.056,350.679,413.412,179.867,17.132,151.686
C02531=1103.050,350.432,413.446,179.863,17.128,151.686
C02532=1103.044,350.184,413.480,179.860,17.126,151.686
C02533=1103.038,349.936,413.514,179.857,17.123,151.686
C02534=1103.033,349.689,413.549,179.854,17.119,151.685
C02535=1103.027,349.441,413.582,179.851,17.116,151.685
C02536=1103.021,349.194,413.616,179.848,17.113,151.685
C02537=1103.016,348.946,413.650,179.844,17.110,151.685
C02538=1103.011,348.698,413.684,179.841,17.107,151.685
C02539=1103.005,348.451,413.718,179.838,17.104,151.685
C02540=1102.998,348.203,413.753,179.835,17.101,151.685
C02541=1102.993,347.955,413.786,179.832,17.098,151.685
C02542=1102.987,347.708,413.820,179.829,17.095,151.685
C02543=1102.981,347.460,413.854,179.825,17.092,151.684
C02544=1102.976,347.212,413.888,179.823,17.089,151.684
C02545=1102.970,346.965,413.922,179.820,17.086,151.684
C02546=1102.965,346.717,413.955,179.816,17.083,151.684
C02547=1102.959,346.470,413.989,179.813,17.080,151.684
C02548=1102.953,346.222,414.023,179.810,17.077,151.684
C02549=1102.948,345.974,414.057,179.807,17.074,151.684
C02550=1102.942,345.727,414.090,179.804,17.071,151.684
C02551=1102.936,345.479,414.124,179.800,17.068,151.684
C02552=1102.931,345.231,414.158,179.798,17.065,151.684
C02553=1102.925,344.984,414.192,179.794,17.062,151.684
C02554=1102.919,344.736,414.225,179.791,17.059,151.683
C02555=1102.913,344.489,414.259,179.788,17.056,151.683
C02556=1102.908,344.241,414.292,179.785,17.054,151.683
C02557=1102.902,343.992,414.326,179.781,17.050,151.683
C02558=1102.893,343.622,414.377,179.777,17.046,151.683
C02559=1102.885,343.252,414.427,179.772,17.042,151.683
C02560=1102.876,342.882,414.477,179.767,17.038,151.683
C02561=1102.868,342.510,414.528,179.762,17.034,151.683
C02562=1102.862,342.264,414.560,179.760,17.031,151.683
C02563=1102.857,342.016,414.594,179.756,17.028,151.683
C02564=1102.851,341.768,414.627,179.753,17.025,151.683
C02565=1102.845,341.521,414.661,179.750,17.022,151.683
C02566=1102.840,341.273,414.694,179.747,17.020,151.683
C02567=1102.834,341.025,414.728,179.743,17.017,151.683
C02568=1102.828,340.777,414.761,179.740,17.014,151.683
C02569=1102.823,340.529,414.794,179.737,17.011,151.683
C02570=1102.817,340.282,414.828,179.734,17.009,151.683
C02571=1102.812,340.034,414.862,179.730,17.005,151.683
C02572=1102.805,339.786,414.895,179.727,17.003,151.683
C02573=1102.800,339.538,414.928,179.724,17.000,151.683
C02574=1102.794,339.290,414.961,179.721,16.997,151.683
C02575=1102.789,339.042,414.995,179.718,16.995,151.683
C02576=1102.783,338.794,415.028,179.714,16.992,151.683
C02577=1102.777,338.547,415.061,179.711,16.989,151.683
C02578=1102.771,338.299,415.094,179.708,16.987,151.683
C02579=1102.766,338.052,415.127,179.705,16.984,151.683
C02580=1102.761,337.804,415.160,179.702,16.982,151.683
C02581=1102.754,337.556,415.193,179.698,16.979,151.683
C02582=1102.749,337.308,415.226,179.695,16.976,151.683
C02583=1102.743,337.060,415.260,179.692,16.973,151.683
C02584=1102.738,336.813,415.293,179.688,16.971,151.683
C02585=1102.731,336.565,415.326,179.685,16.968,151.683
C02586=1102.726,336.317,415.359,179.682,16.966,151.683
C02587=1102.720,336.069,415.392,179.678,16.963,151.683
C02588=1102.715,335.822,415.425,179.675,16.960,151.683
C02589=1102.709,335.574,415.458,179.672,16.958,151.683
C02590=1102.704,335.326,415.491,179.669,16.955,151.683
C02591=1102.697,335.079,415.524,179.666,16.953,151.683
C02592=1102.692,334.830,415.557,179.663,16.950,151.683
C02593=1102.686,334.583,415.590,179.659,16.948,151.683
C02594=1102.680,334.335,415.623,179.656,16.945,151.683
C02595=1102.675,334.088,415.656,179.653,16.942,151.683
C02596=1102.669,333.840,415.689,179.649,16.940,151.683
C02597=1102.664,333.592,415.721,179.646,16.938,151.683
C02598=1102.658,333.344,415.755,179.643,16.935,151.683
C02599=1102.652,333.096,415.787,179.640,16.933,151.683
C02600=1102.647,332.849,415.820,179.637,16.930,151.683
C02601=1102.641,332.601,415.852,179.633,16.927,151.683
C02602=1102.635,332.353,415.886,179.629,16.925,151.684
C02603=1102.629,332.105,415.918,179.626,16.922,151.684
C02604=1102.624,331.857,415.951,179.623,16.920,151.684
C02605=1102.618,331.610,415.983,179.620,16.918,151.684
C02606=1102.612,331.362,416.017,179.617,16.915,151.684
C02607=1102.607,331.114,416.049,179.613,16.913,151.684
C02608=1102.600,330.866,416.082,179.610,16.910,151.684
C02609=1102.595,330.618,416.115,179.607,16.908,151.684
C02610=1102.587,330.241,416.164,179.602,16.905,151.684
C02611=1102.577,329.865,416.213,179.597,16.900,151.684
C02612=1102.568,329.488,416.263,179.592,16.897,151.685
C02613=1102.559,329.112,416.313,179.587,16.894,151.685
C02614=1102.554,328.864,416.344,179.583,16.892,151.685
C02615=1102.548,328.616,416.378,179.580,16.889,151.685
C02616=1102.542,328.368,416.410,179.577,16.887,151.685
C02617=1102.536,328.120,416.442,179.574,16.884,151.685
C02618=1102.531,327.873,416.475,179.570,16.882,151.685
C02619=1102.525,327.624,416.507,179.567,16.880,151.685
C02620=1102.519,327.377,416.539,179.564,16.878,151.685
C02621=1102.514,327.129,416.571,179.561,16.876,151.686
C02622=1102.508,326.881,416.604,179.556,16.873,151.686
C02623=1102.502,326.633,416.636,179.553,16.870,151.686
C02624=1102.496,326.385,416.668,179.550,16.868,151.686
C02625=1102.490,326.138,416.701,179.546,16.866,151.686
C02626=1102.485,325.889,416.733,179.543,16.864,151.686
C02627=1102.479,325.641,416.765,179.540,16.861,151.686
C02628=1102.474,325.394,416.797,179.537,16.859,151.687
C02629=1102.468,325.146,416.830,179.534,16.857,151.687
C02630=1102.463,324.898,416.862,179.530,16.855,151.687
C02631=1102.457,324.650,416.894,179.527,16.853,151.687
C02632=1102.451,324.403,416.927,179.524,16.850,151.687
C02633=1102.445,324.155,416.958,179.520,16.848,151.687
C02634=1102.439,323.907,416.990,179.517,16.846,151.687
C02635=1102.434,323.658,417.023,179.513,16.844,151.688
C02636=1102.429,323.411,417.055,179.510,16.842,151.688
C02637=1102.423,323.163,417.087,179.507,16.839,151.688
C02638=1102.417,322.916,417.119,179.504,16.837,151.688
C02639=1102.411,322.667,417.151,179.500,16.835,151.688
C02640=1102.405,322.419,417.183,179.497,16.833,151.688
C02641=1102.400,322.171,417.215,179.494,16.830,151.688
C02642=1102.394,321.923,417.248,179.490,16.828,151.688
C02643=1102.389,321.676,417.279,179.487,16.826,151.689
C02644=1102.383,321.427,417.311,179.484,16.824,151.689
C02645=1102.378,321.180,417.343,179.480,16.822,151.689
C02646=1102.372,320.932,417.375,179.477,16.820,151.689
C02647=1102.366,320.684,417.407,179.473,16.818,151.689
C02648=1102.360,320.436,417.439,179.470,16.815,151.689
C02649=1102.355,320.188,417.470,179.467,16.813,151.690
C02650=1102.350,319.940,417.503,179.464,16.811,151.690
C02651=1102.344,319.692,417.535,179.460,16.809,151.690
C02652=1102.338,319.444,417.567,179.457,16.807,151.690
C02653=1102.333,319.197,417.598,179.453,16.805,151.690
C02654=1102.327,318.948,417.630,179.450,16.802,151.691
C02655=1102.321,318.701,417.662,179.447,16.800,151.691
C02656=1102.315,318.453,417.694,179.443,16.798,151.691
C02657=1102.310,318.205,417.726,179.441,16.797,151.691
C02658=1102.304,317.957,417.758,179.437,16.795,151.691
C02659=1102.299,317.709,417.789,179.434,16.793,151.691
C02660=1102.294,317.461,417.820,179.431,16.790,151.691
C02661=1102.288,317.213,417.852,179.427,16.788,151.692
C02662=1102.279,316.830,417.901,179.422,16.785,151.692
C02663=1102.271,316.446,417.950,179.416,16.781,151.692
C02664=1102.262,316.063,417.999,179.411,16.778,151.693
C02665=1102.253,315.678,418.049,179.406,16.775,151.693
C02666=1102.248,315.430,418.080,179.403,16.773,151.693
C02667=1102.243,315.183,418.111,179.399,16.771,151.693
C02668=1102.236,314.935,418.143,179.397,16.769,151.693
C02669=1102.231,314.687,418.174,179.393,16.767,151.694
C02670=1102.225,314.438,418.206,179.390,16.766,151.694
C02671=1102.219,314.191,418.237,179.386,16.763,151.694
C02672=1102.213,313.943,418.269,179.383,16.761,151.694
C02673=1102.208,313.695,418.300,179.379,16.760,151.695
C02674=1102.201,313.447,418.331,179.376,16.758,151.695
C02675=1102.196,313.199,418.362,179.372,16.756,151.695
C02676=1102.191,312.951,418.394,179.369,16.754,151.695
C02677=1102.184,312.704,418.425,179.365,16.752,151.696
C02678=1102.179,312.455,418.456,179.362,16.751,151.696
C02679=1102.173,312.207,418.488,179.359,16.748,151.696
C02680=1102.167,311.959,418.518,179.356,16.746,151.696
C02681=1102.162,311.712,418.550,179.352,16.745,151.697
C02682=1102.156,311.463,418.581,179.348,16.743,151.697
C02683=1102.150,311.216,418.613,179.345,16.741,151.697
C02684=1102.144,310.967,418.644,179.341,16.739,151.697
C02685=1102.138,310.720,418.675,179.338,16.737,151.698
C02686=1102.133,310.472,418.706,179.334,16.735,151.698
C02687=1102.127,310.223,418.738,179.332,16.734,151.698
C02688=1102.121,309.976,418.768,179.328,16.732,151.698
C02689=1102.116,309.728,418.800,179.325,16.730,151.699
C02690=1102.109,309.480,418.831,179.321,16.728,151.699
C02691=1102.104,309.231,418.862,179.318,16.726,151.699
C02692=1102.098,308.984,418.893,179.314,16.724,151.700
C02693=1102.093,308.736,418.924,179.310,16.722,151.700
C02694=1102.087,308.488,418.954,179.308,16.721,151.700
C02695=1102.081,308.240,418.986,179.304,16.719,151.700
C02696=1102.076,307.992,419.017,179.301,16.717,151.701
C02697=1102.070,307.743,419.048,179.297,16.715,151.701
C02698=1102.064,307.496,419.079,179.293,16.714,151.701
C02699=1102.059,307.248,419.110,179.290,16.711,151.701
C02700=1102.053,307.000,419.141,179.286,16.710,151.702
C02701=1102.047,306.753,419.172,179.283,16.708,151.702
C02702=1102.042,306.504,419.203,179.280,16.707,151.702
C02703=1102.036,306.256,419.233,179.277,16.705,151.702
C02704=1102.031,306.008,419.264,179.273,16.703,151.703
C02705=1102.025,305.760,419.295,179.270,16.701,151.703
C02706=1102.018,305.512,419.326,179.266,16.699,151.703
C02707=1102.013,305.264,419.357,179.262,16.697,151.704
C02708=1102.007,305.016,419.387,179.259,16.695,151.704
C02709=1102.002,304.768,419.418,179.256,16.694,151.704
C02710=1101.996,304.520,419.449,179.253,16.692,151.704
C02711=1101.991,304.272,419.480,179.249,16.690,151.705
C02712=1101.985,304.024,419.510,179.245,16.689,151.705
C02713=1101.979,303.776,419.541,179.242,16.687,151.705
C02714=1101.971,303.395,419.589,179.236,16.684,151.706
C02715=1101.963,303.014,419.636,179.231,16.681,151.706
C02716=1101.954,302.632,419.683,179.226,16.679,151.707
C02717=1101.945,302.252,419.729,179.221,16.676,151.707
C02718=1101.939,302.003,419.760,179.217,16.675,151.707
C02719=1101.934,301.755,419.791,179.214,16.673,151.708
C02720=1101.928,301.507,419.822,179.210,16.671,151.708
C02721=1101.923,301.259,419.852,179.207,16.669,151.708
C02722=1101.917,301.012,419.882,179.204,16.668,151.708
C02723=1101.912,300.763,419.913,179.200,16.666,151.709
C02724=1101.906,300.516,419.944,179.197,16.664,151.709
C02725=1101.900,300.268,419.974,179.193,16.662,151.709
C02726=1101.895,300.020,420.005,179.190,16.661,151.710
C02727=1101.890,299.771,420.034,179.187,16.660,151.710
C02728=1101.884,299.523,420.065,179.183,16.657,151.710
C02729=1101.879,299.275,420.096,179.180,16.656,151.711
C02730=1101.873,299.027,420.126,179.176,16.654,151.711
C02731=1101.867,298.780,420.156,179.172,16.652,151.711
C02732=1101.861,298.532,420.187,179.170,16.651,151.712
C02733=1101.856,298.283,420.217,179.166,16.649,151.712
C02734=1101.851,298.035,420.247,179.162,16.648,151.712
C02735=1101.845,297.787,420.278,179.159,16.646,151.713
C02736=1101.839,297.540,420.308,179.155,16.644,151.713
C02737=1101.833,297.291,420.338,179.152,16.643,151.713
C02738=1101.828,297.043,420.368,179.149,16.641,151.713
C02739=1101.822,296.796,420.398,179.145,16.639,151.714
C02740=1101.817,296.547,420.429,179.141,16.638,151.714
C02741=1101.811,296.299,420.459,179.138,16.637,151.715
C02742=1101.805,296.050,420.490,179.135,16.635,151.715
C02743=1101.799,295.802,420.519,179.131,16.633,151.715
C02744=1101.793,295.554,420.550,179.127,16.632,151.716
C02745=1101.788,295.306,420.580,179.124,16.631,151.716
C02746=1101.782,295.058,420.610,179.121,16.629,151.716
C02747=1101.776,294.810,420.640,179.117,16.627,151.717
C02748=1101.771,294.562,420.670,179.113,16.626,151.717
C02749=1101.765,294.314,420.700,179.110,16.625,151.717
C02750=1101.760,294.065,420.730,179.107,16.623,151.718
C02751=1101.754,293.818,420.760,179.103,16.621,151.718
C02752=1101.749,293.570,420.789,179.099,16.620,151.718
C02753=1101.743,293.322,420.820,179.096,16.619,151.719
C02754=1101.737,293.074,420.849,179.093,16.617,151.719
C02755=1101.732,292.826,420.880,179.089,16.615,151.720
C02756=1101.726,292.577,420.909,179.085,16.614,151.720
C02757=1101.720,292.329,420.940,179.082,16.613,151.720
C02758=1101.715,292.081,420.969,179.079,16.611,151.721
C02759=1101.708,291.833,420.999,179.075,16.609,151.721
C02760=1101.703,291.585,421.029,179.072,16.608,151.721
C02761=1101.697,291.337,421.058,179.068,16.606,151.722
C02762=1101.691,291.089,421.089,179.065,16.605,151.722
C02763=1101.686,290.840,421.118,179.061,16.603,151.722
C02764=1101.680,290.592,421.148,179.058,16.602,151.723
C02765=1101.675,290.344,421.178,179.054,16.600,151.723
C02766=1101.667,289.977,421.222,179.050,16.599,151.724
C02767=1101.658,289.609,421.266,179.044,16.596,151.724
C02768=1101.650,289.243,421.310,179.039,16.595,151.725
C02769=1101.641,288.875,421.353,179.034,16.592,151.725
C02770=1101.635,288.627,421.383,179.030,16.590,151.726
C02771=1101.629,288.379,421.413,179.027,16.589,151.726
C02772=1101.624,288.130,421.443,179.023,16.588,151.727
C02773=1101.618,287.883,421.472,179.019,16.587,151.727
C02774=1101.613,287.635,421.501,179.016,16.585,151.727
C02775=1101.607,287.386,421.531,179.013,16.584,151.728
C02776=1101.602,287.138,421.561,179.009,16.583,151.728
C02777=1101.595,286.890,421.590,179.006,16.582,151.729
C02778=1101.590,286.642,421.620,179.002,16.580,151.729
C02779=1101.584,286.393,421.650,178.998,16.578,151.729
C02780=1101.578,286.146,421.678,178.995,16.577,151.730
C02781=1101.573,285.897,421.708,178.991,16.576,151.730
C02782=1101.567,285.649,421.738,178.988,16.574,151.731
C02783=1101.561,285.401,421.767,178.985,16.573,151.731
C02784=1101.556,285.152,421.796,178.981,16.572,151.731
C02785=1101.551,284.905,421.826,178.977,16.570,151.732
C02786=1101.545,284.657,421.855,178.974,16.569,151.732
C02787=1101.539,284.408,421.884,178.971,16.568,151.733
C02788=1101.534,284.160,421.914,178.967,16.566,151.733
C02789=1101.527,283.912,421.943,178.964,16.565,151.733
C02790=1101.522,283.664,421.972,178.960,16.564,151.734
C02791=1101.517,283.415,422.002,178.956,16.562,151.734
C02792=1101.511,283.167,422.031,178.953,16.561,151.734
C02793=1101.505,282.919,422.060,178.949,16.560,151.735
C02794=1101.499,282.671,422.089,178.946,16.558,151.735
C02795=1101.494,282.423,422.119,178.943,16.557,151.736
C02796=1101.488,282.174,422.148,178.939,16.555,151.736
C02797=1101.482,281.926,422.177,178.935,16.554,151.737
C02798=1101.478,281.678,422.206,178.932,16.553,151.737
C02799=1101.471,281.430,422.235,178.929,16.552,151.737
C02800=1101.466,281.181,422.265,178.925,16.550,151.738
C02801=1101.460,280.934,422.293,178.922,16.549,151.738
C02802=1101.455,280.686,422.323,178.918,16.548,151.739
C02803=1101.449,280.437,422.351,178.915,16.547,151.739
C02804=1101.443,280.188,422.381,178.911,16.545,151.739
C02805=1101.438,279.941,422.410,178.907,16.544,151.740
C02806=1101.432,279.692,422.439,178.904,16.543,151.740
C02807=1101.426,279.444,422.468,178.900,16.542,151.741
C02808=1101.421,279.195,422.497,178.896,16.540,151.741
C02809=1101.415,278.948,422.526,178.894,16.539,151.742
C02810=1101.409,278.699,422.554,178.890,16.538,151.742
C02811=1101.403,278.451,422.584,178.887,16.537,151.742
C02812=1101.398,278.203,422.612,178.883,16.536,151.743
C02813=1101.393,277.954,422.641,178.879,16.534,151.743
C02814=1101.386,277.706,422.670,178.876,16.533,151.744
C02815=1101.381,277.459,422.699,178.872,16.532,151.744
C02816=1101.376,277.210,422.728,178.869,16.531,151.745
C02817=1101.369,276.961,422.757,178.865,16.530,151.745
C02818=1101.362,276.604,422.798,178.860,16.528,151.746
C02819=1101.353,276.246,422.839,178.855,16.526,151.746
C02820=1101.345,275.888,422.882,178.849,16.524,151.747
C02821=1101.337,275.530,422.923,178.845,16.522,151.748
C02822=1101.331,275.281,422.952,178.841,16.522,151.748
C02823=1101.326,275.033,422.980,178.838,16.520,151.749
C02824=1101.320,274.785,423.009,178.834,16.519,151.749
C02825=1101.315,274.537,423.037,178.831,16.518,151.749
C02826=1101.309,274.289,423.066,178.827,16.517,151.750
C02827=1101.303,274.040,423.095,178.824,16.516,151.750
C02828=1101.298,273.792,423.123,178.820,16.514,151.751
C02829=1101.292,273.544,423.152,178.816,16.513,151.751
C02830=1101.286,273.296,423.180,178.813,16.512,151.752
C02831=1101.280,273.047,423.209,178.809,16.510,151.752
C02832=1101.275,272.798,423.238,178.806,16.510,151.753
C02833=1101.270,272.550,423.266,178.802,16.508,151.753
C02834=1101.263,272.302,423.295,178.799,16.508,151.754
C02835=1101.258,272.054,423.323,178.795,16.506,151.754
C02836=1101.252,271.805,423.352,178.792,16.505,151.754
C02837=1101.246,271.558,423.380,178.788,16.504,151.755
C02838=1101.241,271.309,423.409,178.785,16.503,151.755
C02839=1101.236,271.061,423.437,178.781,16.502,151.756
C02840=1101.230,270.812,423.465,178.777,16.501,151.756
C02841=1101.224,270.564,423.494,178.775,16.500,151.757
C02842=1101.218,270.316,423.522,178.771,16.498,151.757
C02843=1101.212,270.067,423.551,178.767,16.497,151.758
C02844=1101.207,269.819,423.579,178.764,16.496,151.758
C02845=1101.201,269.570,423.607,178.760,16.495,151.759
C02846=1101.196,269.323,423.636,178.757,16.494,151.759
C02847=1101.190,269.074,423.664,178.753,16.493,151.760
C02848=1101.184,268.826,423.692,178.750,16.492,151.760
C02849=1101.178,268.577,423.720,178.746,16.491,151.760
C02850=1101.173,268.329,423.748,178.743,16.490,151.761
C02851=1101.167,268.081,423.777,178.739,16.489,151.762
C02852=1101.162,267.832,423.805,178.736,16.488,151.762
C02853=1101.155,267.584,423.834,178.732,16.487,151.762
C02854=1101.150,267.336,423.862,178.728,16.485,151.763
C02855=1101.144,267.088,423.890,178.725,16.484,151.763
C02856=1101.139,266.840,423.918,178.721,16.483,151.764
C02857=1101.133,266.591,423.946,178.718,16.482,151.764
C02858=1101.127,266.343,423.974,178.714,16.481,151.765
C02859=1101.122,266.094,424.002,178.711,16.480,151.765
C02860=1101.116,265.846,424.030,178.707,16.479,151.766
C02861=1101.111,265.598,424.058,178.704,16.478,151.766
C02862=1101.105,265.349,424.087,178.700,16.477,151.767
C02863=1101.100,265.101,424.115,178.697,16.476,151.767
C02864=1101.094,264.852,424.142,178.693,16.475,151.768
C02865=1101.089,264.604,424.170,178.690,16.474,151.768
C02866=1101.083,264.356,424.198,178.686,16.473,151.769
C02867=1101.077,264.107,424.227,178.682,16.472,151.769
C02868=1101.071,263.859,424.254,178.678,16.471,151.770
C02869=1101.065,263.610,424.282,178.675,16.470,151.770
C02870=1101.057,263.255,424.322,178.670,16.469,151.771
C02871=1101.049,262.899,424.362,178.665,16.468,151.772
C02872=1101.040,262.545,424.402,178.660,16.466,151.772
C02873=1101.032,262.190,424.442,178.655,16.465,151.773
C02874=1101.027,261.941,424.469,178.651,16.464,151.774
C02875=1101.021,261.693,424.497,178.648,16.463,151.774
C02876=1101.015,261.445,424.525,178.644,16.461,151.775
C02877=1101.009,261.196,424.553,178.641,16.461,151.775
C02878=1101.004,260.948,424.580,178.637,16.460,151.776
C02879=1100.998,260.699,424.608,178.634,16.459,151.776
C02880=1100.992,260.451,424.636,178.630,16.458,151.777
C02881=1100.987,260.203,424.664,178.626,16.457,151.777
C02882=1100.981,259.954,424.691,178.622,16.456,151.778
C02883=1100.975,259.706,424.719,178.619,16.455,151.778
C02884=1100.970,259.458,424.747,178.615,16.454,151.779
C02885=1100.964,259.209,424.774,178.612,16.453,151.779
C02886=1100.958,258.961,424.802,178.608,16.452,151.780
C02887=1100.952,258.712,424.828,178.605,16.451,151.780
C02888=1100.947,258.464,424.857,178.601,16.450,151.781
C02889=1100.941,258.216,424.885,178.598,16.450,151.781
C02890=1100.935,257.967,424.911,178.594,16.448,151.782
C02891=1100.929,257.718,424.940,178.591,16.447,151.782
C02892=1100.924,257.470,424.967,178.587,16.446,151.783
C02893=1100.918,257.222,424.994,178.584,16.446,151.783
C02894=1100.913,256.973,425.022,178.580,16.445,151.784
C02895=1100.907,256.725,425.049,178.576,16.444,151.784
C02896=1100.902,256.476,425.076,178.572,16.443,151.785
C02897=1100.896,256.228,425.104,178.569,16.442,151.785
C02898=1100.890,255.979,425.131,178.565,16.441,151.786
C02899=1100.885,255.731,425.159,178.562,16.440,151.786
C02900=1100.879,255.483,425.186,178.559,16.439,151.787
C02901=1100.873,255.234,425.214,178.555,16.438,151.787
C02902=1100.867,254.986,425.241,178.552,16.438,151.788
C02903=1100.862,254.737,425.268,178.548,16.436,151.788
C02904=1100.856,254.489,425.296,178.545,16.436,151.789
C02905=1100.851,254.241,425.323,178.541,16.435,151.790
C02906=1100.845,253.991,425.350,178.537,16.434,151.790
C02907=1100.839,253.743,425.378,178.534,16.432,151.790
C02908=1100.833,253.495,425.404,178.530,16.432,151.791
C02909=1100.828,253.246,425.432,178.526,16.431,151.792
C02910=1100.822,252.999,425.459,178.523,16.430,151.792
C02911=1100.817,252.749,425.487,178.520,16.430,151.793
C02912=1100.811,252.501,425.513,178.516,16.428,151.793
C02913=1100.806,252.252,425.541,178.513,16.428,151.794
C02914=1100.800,252.004,425.568,178.509,16.427,151.794
C02915=1100.795,251.756,425.595,178.506,16.426,151.795
C02916=1100.789,251.507,425.622,178.502,16.424,151.795
C02917=1100.783,251.258,425.649,178.499,16.424,151.796
C02918=1100.777,251.010,425.677,178.495,16.423,151.796
C02919=1100.772,250.762,425.704,178.491,16.422,151.797
C02920=1100.766,250.513,425.731,178.488,16.422,151.797
C02921=1100.761,250.265,425.758,178.484,16.420,151.798
C02922=1100.753,249.907,425.797,178.479,16.419,151.799
C02923=1100.745,249.548,425.835,178.474,16.418,151.799
C02924=1100.737,249.191,425.874,178.469,16.416,151.800
C02925=1100.730,248.833,425.914,178.464,16.415,151.801
C02926=1100.723,248.584,425.941,178.461,16.414,151.801
C02927=1100.717,248.336,425.967,178.457,16.413,151.802
C02928=1100.712,248.087,425.995,178.453,16.413,151.802
C02929=1100.707,247.839,426.021,178.450,16.412,151.803
C02930=1100.702,247.590,426.048,178.446,16.411,151.803
C02931=1100.696,247.342,426.075,178.443,16.410,151.804
C02932=1100.690,247.093,426.102,178.439,16.409,151.804
C02933=1100.684,246.845,426.128,178.436,16.408,151.805
C02934=1100.679,246.596,426.156,178.433,16.408,151.806
C02935=1100.673,246.348,426.182,178.429,16.407,151.806
C02936=1100.668,246.100,426.209,178.425,16.406,151.807
C02937=1100.662,245.851,426.236,178.421,16.405,151.807
C02938=1100.656,245.602,426.261,178.418,16.404,151.808
C02939=1100.651,245.354,426.289,178.415,16.404,151.808
C02940=1100.646,245.105,426.315,178.411,16.403,151.809
C02941=1100.639,244.856,426.342,178.408,16.402,151.809
C02942=1100.633,244.608,426.369,178.404,16.401,151.810
C02943=1100.628,244.359,426.396,178.400,16.400,151.810
C02944=1100.623,244.111,426.423,178.397,16.400,151.811
C02945=1100.617,243.862,426.449,178.393,16.399,151.812
C02946=1100.611,243.613,426.476,178.390,16.398,151.812
C02947=1100.606,243.365,426.502,178.386,16.397,151.813
C02948=1100.600,243.117,426.529,178.383,16.396,151.813
C02949=1100.594,242.868,426.555,178.379,16.396,151.814
C02950=1100.589,242.619,426.581,178.375,16.395,151.814
C02951=1100.583,242.371,426.608,178.372,16.394,151.815
C02952=1100.578,242.122,426.635,178.369,16.393,151.815
C02953=1100.572,241.874,426.662,178.365,16.392,151.816
C02954=1100.567,241.625,426.688,178.362,16.392,151.816
C02955=1100.561,241.377,426.715,178.357,16.391,151.817
C02956=1100.555,241.128,426.741,178.354,16.390,151.818
C02957=1100.550,240.879,426.767,178.351,16.390,151.818
C02958=1100.544,240.631,426.794,178.347,16.389,151.819
C02959=1100.538,240.383,426.820,178.344,16.388,151.819
C02960=1100.533,240.134,426.846,178.341,16.388,151.820
C02961=1100.527,239.885,426.873,178.337,16.386,151.820
C02962=1100.521,239.636,426.899,178.333,16.386,151.821
C02963=1100.515,239.388,426.925,178.329,16.385,151.821
C02964=1100.509,239.140,426.952,178.326,16.384,151.822
C02965=1100.504,238.892,426.977,178.323,16.384,151.823
C02966=1100.498,238.643,427.004,178.319,16.383,151.823
C02967=1100.493,238.394,427.030,178.315,16.382,151.824
C02968=1100.487,238.146,427.056,178.312,16.382,151.824
C02969=1100.482,237.897,427.082,178.308,16.381,151.825
C02970=1100.476,237.649,427.109,178.305,16.380,151.825
C02971=1100.470,237.400,427.135,178.302,16.380,151.826
C02972=1100.465,237.151,427.162,178.298,16.378,151.826
C02973=1100.459,236.902,427.188,178.294,16.378,151.827
C02974=1100.451,236.538,427.226,178.289,16.377,151.828
C02975=1100.442,236.173,427.264,178.284,16.376,151.829
C02976=1100.434,235.808,427.302,178.279,16.375,151.830
C02977=1100.426,235.443,427.340,178.273,16.373,151.830
C02978=1100.420,235.195,427.367,178.270,16.373,151.831
C02979=1100.415,234.946,427.393,178.267,16.373,151.832
C02980=1100.409,234.697,427.419,178.263,16.371,151.832
C02981=1100.404,234.449,427.445,178.259,16.371,151.833
C02982=1100.397,234.200,427.471,178.256,16.370,151.833
C02983=1100.393,233.952,427.496,178.252,16.369,151.834
C02984=1100.387,233.704,427.523,178.249,16.369,151.834
C02985=1100.381,233.455,427.549,178.246,16.368,151.835
C02986=1100.375,233.206,427.574,178.241,16.367,151.835
C02987=1100.369,232.957,427.601,178.238,16.367,151.836
C02988=1100.365,232.709,427.626,178.235,16.366,151.837
C02989=1100.359,232.460,427.652,178.231,16.365,151.837
C02990=1100.353,232.212,427.678,178.228,16.365,151.838
C02991=1100.347,231.963,427.704,178.225,16.364,151.838
C02992=1100.342,231.714,427.730,178.221,16.364,151.839
C02993=1100.337,231.466,427.756,178.217,16.363,151.839
C02994=1100.331,231.217,427.781,178.214,16.362,151.840
C02995=1100.325,230.968,427.807,178.211,16.362,151.841
C02996=1100.320,230.719,427.833,178.207,16.361,151.841
C02997=1100.313,230.471,427.858,178.203,16.360,151.842
C02998=1100.308,230.223,427.885,178.200,16.359,151.842
C02999=1100.303,229.974,427.911,178.196,16.359,151.843
C03000=1100.297,229.725,427.936,178.193,16.358,151.843
C03001=1100.291,229.476,427.962,178.189,16.358,151.844
C03002=1100.285,229.228,427.987,178.186,16.357,151.845
C03003=1100.280,228.979,428.013,178.182,16.356,151.845
C03004=1100.274,228.731,428.038,178.179,16.356,151.846
C03005=1100.268,228.482,428.064,178.175,16.355,151.846
C03006=1100.262,228.233,428.089,178.171,16.354,151.847
C03007=1100.257,227.985,428.115,178.168,16.354,151.847
C03008=1100.251,227.736,428.140,178.165,16.353,151.848
C03009=1100.246,227.487,428.166,178.161,16.353,151.849
C03010=1100.241,227.239,428.192,178.157,16.352,151.849
C03011=1100.235,226.990,428.217,178.154,16.351,151.850
C03012=1100.229,226.741,428.243,178.151,16.351,151.850
C03013=1100.223,226.493,428.268,178.147,16.350,151.851
C03014=1100.218,226.244,428.294,178.143,16.350,151.852
C03015=1100.212,225.996,428.319,178.140,16.349,151.852
C03016=1100.206,225.747,428.345,178.137,16.348,151.853
C03017=1100.201,225.499,428.370,178.133,16.347,151.853
C03018=1100.195,225.249,428.395,178.130,16.347,151.854
C03019=1100.189,225.000,428.421,178.126,16.347,151.854
C03020=1100.184,224.752,428.446,178.122,16.346,151.855
C03021=1100.178,224.503,428.472,178.119,16.345,151.856
C03022=1100.172,224.255,428.497,178.116,16.344,151.856
C03023=1100.167,224.007,428.522,178.112,16.344,151.857
C03024=1100.161,223.757,428.547,178.108,16.343,151.857
C03025=1100.156,223.508,428.573,178.105,16.343,151.858
C03026=1100.147,223.136,428.611,178.099,16.342,151.859
C03027=1100.139,222.762,428.649,178.094,16.341,151.860
C03028=1100.130,222.390,428.686,178.089,16.340,151.861
C03029=1100.122,222.016,428.724,178.084,16.339,151.861
C03030=1100.116,221.767,428.750,178.080,16.338,151.862
C03031=1100.111,221.518,428.774,178.077,16.338,151.863
C03032=1100.105,221.270,428.800,178.074,16.338,151.863
C03033=1100.099,221.021,428.826,178.070,16.337,151.864
C03034=1100.094,220.772,428.850,178.066,16.336,151.864
C03035=1100.088,220.523,428.875,178.063,16.336,151.865
C03036=1100.082,220.275,428.900,178.059,16.335,151.866
C03037=1100.077,220.026,428.925,178.056,16.335,151.866
C03038=1100.071,219.777,428.951,178.052,16.334,151.867
C03039=1100.065,219.529,428.976,178.049,16.334,151.867
C03040=1100.059,219.280,429.000,178.045,16.333,151.868
C03041=1100.054,219.032,429.025,178.042,16.333,151.868
C03042=1100.049,218.782,429.050,178.039,16.332,151.869
C03043=1100.043,218.534,429.075,178.035,16.331,151.870
C03044=1100.037,218.285,429.100,178.031,16.331,151.870
C03045=1100.031,218.036,429.125,178.028,16.330,151.871
C03046=1100.026,217.788,429.150,178.025,16.330,151.872
C03047=1100.020,217.539,429.176,178.021,16.329,151.872
C03048=1100.015,217.290,429.200,178.017,16.329,151.873
C03049=1100.009,217.041,429.225,178.014,16.328,151.873
C03050=1100.003,216.793,429.249,178.011,16.328,151.874
C03051=1099.997,216.544,429.275,178.007,16.327,151.874
C03052=1099.992,216.296,429.299,178.003,16.326,151.875
C03053=1099.986,216.047,429.325,178.000,16.326,151.876
C03054=1099.981,215.798,429.349,177.997,16.325,151.876
C03055=1099.975,215.549,429.374,177.993,16.325,151.877
C03056=1099.970,215.301,429.399,177.989,16.324,151.877
C03057=1099.964,215.052,429.423,177.986,16.323,151.878
C03058=1099.958,214.803,429.448,177.983,16.323,151.879
C03059=1099.953,214.555,429.473,177.979,16.323,151.879
C03060=1099.948,214.305,429.498,177.976,16.322,151.880
C03061=1099.942,214.057,429.522,177.972,16.321,151.880
C03062=1099.936,213.808,429.547,177.969,16.321,151.881
C03063=1099.931,213.559,429.572,177.965,16.321,151.882
C03064=1099.925,213.310,429.596,177.962,16.320,151.882
C03065=1099.919,213.062,429.621,177.959,16.320,151.883
C03066=1099.914,212.814,429.646,177.955,16.318,151.883
C03067=1099.908,212.564,429.670,177.951,16.318,151.884
C03068=1099.903,212.316,429.694,177.948,16.318,151.885
C03069=1099.897,212.067,429.720,177.945,16.317,151.885
C03070=1099.891,211.819,429.744,177.941,16.317,151.886
C03071=1099.885,211.569,429.769,177.937,16.316,151.886
C03072=1099.880,211.321,429.793,177.934,16.316,151.887
C03073=1099.875,211.072,429.817,177.931,16.315,151.887
C03074=1099.869,210.823,429.843,177.927,16.315,151.888
C03075=1099.863,210.575,429.867,177.924,16.315,151.889
C03076=1099.857,210.326,429.891,177.921,16.314,151.889
C03077=1099.851,210.077,429.915,177.916,16.313,151.890
C03078=1099.843,209.708,429.951,177.912,16.313,151.891
C03079=1099.835,209.338,429.987,177.907,16.312,151.892
C03080=1099.827,208.968,430.024,177.901,16.311,151.893
C03081=1099.818,208.600,430.060,177.896,16.310,151.893
C03082=1099.795,207.591,430.158,177.856,16.298,151.899
C03083=1099.790,207.343,430.182,177.853,16.298,151.900
C03084=1099.784,207.094,430.206,177.849,16.299,151.901
C03085=1099.778,206.845,430.230,177.845,16.299,151.902
C03086=1099.773,206.596,430.255,177.841,16.300,151.902
C03087=1099.767,206.348,430.278,177.837,16.300,151.903
C03088=1099.761,206.099,430.303,177.834,16.301,151.904
C03089=1099.756,205.850,430.327,177.831,16.301,151.905
C03090=1099.750,205.601,430.350,177.827,16.301,151.906
C03091=1099.745,205.353,430.374,177.823,16.302,151.907
C03092=1099.739,205.104,430.399,177.819,16.302,151.907
C03093=1099.733,204.855,430.423,177.816,16.302,151.908
C03094=1099.728,204.606,430.446,177.812,16.302,151.909
C03095=1099.722,204.357,430.470,177.808,16.302,151.910
C03096=1099.716,204.109,430.494,177.805,16.303,151.911
C03097=1099.710,203.860,430.519,177.801,16.304,151.911
C03098=1099.705,203.611,430.542,177.797,16.304,151.912
C03099=1099.699,203.362,430.566,177.794,16.304,151.913
C03100=1099.694,203.114,430.590,177.790,16.304,151.914
C03101=1099.689,202.865,430.614,177.786,16.305,151.915
C03102=1099.683,202.616,430.638,177.783,16.305,151.916
C03103=1099.676,202.367,430.661,177.780,16.306,151.916
C03104=1099.671,202.119,430.686,177.776,16.306,151.917
C03105=1099.665,201.870,430.709,177.772,16.307,151.918
C03106=1099.660,201.621,430.733,177.768,16.307,151.919
C03107=1099.654,201.372,430.757,177.765,16.307,151.920
C03108=1099.649,201.123,430.780,177.761,16.307,151.921
C03109=1099.642,200.875,430.804,177.757,16.308,151.921
C03110=1099.637,200.625,430.828,177.754,16.308,151.922
C03111=1099.631,200.377,430.852,177.750,16.309,151.923
C03112=1099.625,200.128,430.875,177.746,16.309,151.924
C03113=1099.620,199.879,430.899,177.743,16.310,151.925
C03114=1099.614,199.631,430.923,177.739,16.310,151.926
C03115=1099.608,199.381,430.946,177.735,16.310,151.926
C03116=1099.602,199.133,430.970,177.731,16.310,151.927
C03117=1099.596,198.884,430.993,177.729,16.311,151.928
C03118=1099.591,198.635,431.017,177.725,16.311,151.929
C03119=1099.585,198.386,431.040,177.721,16.312,151.930
C03120=1099.580,198.138,431.065,177.717,16.312,151.930
C03121=1099.574,197.888,431.088,177.714,16.312,151.931
C03122=1099.568,197.640,431.112,177.710,16.312,151.932
C03123=1099.563,197.391,431.135,177.707,16.313,151.933
C03124=1099.557,197.142,431.159,177.703,16.313,151.934
C03125=1099.551,196.893,431.182,177.700,16.313,151.934
C03126=1099.546,196.644,431.205,177.696,16.314,151.935
C03127=1099.540,196.396,431.229,177.692,16.314,151.936
C03128=1099.534,196.147,431.252,177.688,16.314,151.937
C03129=1099.529,195.899,431.276,177.685,16.315,151.938
C03130=1099.523,195.649,431.299,177.682,16.315,151.938
C03131=1099.517,195.400,431.322,177.678,16.316,151.939
C03132=1099.512,195.151,431.347,177.674,16.316,151.940
C03133=1099.506,194.903,431.370,177.671,16.316,151.941
C03134=1099.500,194.654,431.392,177.667,16.316,151.942
C03135=1099.495,194.405,431.417,177.663,16.316,151.943
C03136=1099.489,194.156,431.440,177.660,16.317,151.943
C03137=1099.483,193.907,431.463,177.657,16.317,151.944
C03138=1099.478,193.658,431.486,177.653,16.318,151.945
C03139=1099.472,193.410,431.510,177.649,16.318,151.946
C03140=1099.467,193.161,431.533,177.645,16.318,151.947
C03141=1099.461,192.912,431.556,177.642,16.318,151.947
C03142=1099.456,192.663,431.579,177.639,16.319,151.948
C03143=1099.449,192.389,431.605,177.635,16.319,151.949
C03144=1099.443,192.117,431.630,177.631,16.319,151.950
C03145=1099.437,191.843,431.655,177.627,16.319,151.951
C03146=1099.430,191.570,431.681,177.623,16.320,151.952
C03147=1099.425,191.320,431.705,177.619,16.320,151.952
C03148=1099.419,191.071,431.728,177.616,16.321,151.953
C03149=1099.414,190.822,431.751,177.613,16.321,151.954
C03150=1099.408,190.575,431.774,177.609,16.321,151.955
C03151=1099.403,190.326,431.797,177.605,16.321,151.955
C03152=1099.398,190.077,431.821,177.601,16.322,151.956
C03153=1099.392,189.828,431.844,177.598,16.322,151.957
C03154=1099.386,189.579,431.867,177.595,16.322,151.958
C03155=1099.380,189.330,431.890,177.591,16.323,151.959
C03156=1099.375,189.081,431.912,177.588,16.323,151.959
C03157=1099.370,188.832,431.936,177.584,16.323,151.960
C03158=1099.364,188.583,431.959,177.580,16.323,151.961
C03159=1099.358,188.334,431.982,177.577,16.323,151.962
C03160=1099.352,188.085,432.005,177.574,16.324,151.963
C03161=1099.347,187.836,432.028,177.570,16.324,151.963
C03162=1099.341,187.588,432.051,177.567,16.324,151.964
C03163=1099.337,187.339,432.074,177.563,16.324,151.965
C03164=1099.331,187.090,432.097,177.559,16.324,151.966
C03165=1099.325,186.841,432.120,177.557,16.325,151.966
C03166=1099.319,186.592,432.143,177.553,16.325,151.967
C03167=1099.314,186.343,432.166,177.549,16.325,151.968
C03168=1099.308,186.095,432.189,177.546,16.325,151.969
C03169=1099.302,185.846,432.212,177.542,16.325,151.969
C03170=1099.297,185.596,432.235,177.539,16.325,151.970
C03171=1099.292,185.348,432.257,177.536,16.326,151.971
C03172=1099.287,185.099,432.280,177.532,16.326,151.972
C03173=1099.281,184.850,432.303,177.528,16.326,151.972
C03174=1099.274,184.601,432.325,177.525,16.327,151.973
C03175=1099.269,184.352,432.348,177.521,16.327,151.974
C03176=1099.263,184.103,432.371,177.518,16.328,151.975
C03177=1099.257,183.855,432.394,177.514,16.328,151.975
C03178=1099.252,183.606,432.417,177.511,16.328,151.976
C03179=1099.246,183.356,432.439,177.507,16.328,151.977
C03180=1099.240,183.108,432.462,177.504,16.329,151.978
C03181=1099.234,182.859,432.485,177.500,16.329,151.979
C03182=1099.228,182.610,432.507,177.497,16.329,151.979
C03183=1099.222,182.361,432.530,177.493,16.329,151.980
C03184=1099.218,182.112,432.552,177.489,16.330,151.981
C03185=1099.211,181.863,432.575,177.487,16.330,151.982
C03186=1099.205,181.615,432.598,177.483,16.330,151.982
C03187=1099.200,181.366,432.621,177.479,16.331,151.983
C03188=1099.194,181.116,432.643,177.476,16.331,151.984
C03189=1099.188,180.868,432.665,177.472,16.331,151.985
C03190=1099.182,180.619,432.688,177.469,16.332,151.986
C03191=1099.177,180.369,432.710,177.466,16.332,151.986
C03192=1099.171,180.121,432.733,177.462,16.332,151.987
C03193=1099.166,179.872,432.756,177.459,16.332,151.988
C03194=1099.160,179.623,432.777,177.455,16.333,151.989
C03195=1099.154,179.374,432.800,177.452,16.333,151.989
C03196=1099.148,179.125,432.823,177.448,16.333,151.990
C03197=1099.142,178.876,432.845,177.445,16.333,151.991
C03198=1099.137,178.628,432.868,177.441,16.333,151.992
C03199=1099.131,178.378,432.890,177.438,16.334,151.992
C03200=1099.126,178.129,432.913,177.435,16.334,151.993
C03201=1099.119,177.881,432.935,177.431,16.334,151.994
C03202=1099.114,177.631,432.957,177.427,16.334,151.995
C03203=1099.109,177.383,432.980,177.425,16.335,151.995
C03204=1099.103,177.134,433.002,177.421,16.335,151.996
C03205=1099.097,176.885,433.024,177.417,16.335,151.997
C03206=1099.091,176.635,433.047,177.414,16.335,151.998
C03207=1099.085,176.362,433.071,177.410,16.335,151.998
C03208=1099.079,176.088,433.096,177.407,16.335,151.999
C03209=1099.073,175.815,433.120,177.403,16.336,152.000
C03210=1099.066,175.541,433.144,177.399,16.336,152.001
C03211=1099.061,175.291,433.167,177.395,16.336,152.002
C03212=1099.055,175.043,433.189,177.393,16.337,152.002
C03213=1099.049,174.794,433.211,177.389,16.337,152.003
C03214=1099.044,174.545,433.234,177.385,16.337,152.004
C03215=1099.039,174.296,433.256,177.382,16.337,152.005
C03216=1099.032,174.048,433.278,177.378,16.337,152.005
C03217=1099.027,173.798,433.300,177.376,16.337,152.006
C03218=1099.021,173.550,433.322,177.372,16.337,152.007
C03219=1099.016,173.301,433.345,177.368,16.337,152.007
C03220=1099.010,173.051,433.367,177.365,16.337,152.008
C03221=1099.004,172.802,433.388,177.362,16.338,152.009
C03222=1098.999,172.554,433.411,177.359,16.338,152.010
C03223=1098.993,172.304,433.433,177.355,16.338,152.010
C03224=1098.987,172.055,433.455,177.351,16.338,152.011
C03225=1098.982,171.807,433.477,177.349,16.339,152.012
C03226=1098.976,171.558,433.499,177.345,16.339,152.012
C03227=1098.971,171.309,433.521,177.342,16.339,152.013
C03228=1098.965,171.060,433.543,177.338,16.339,152.014
C03229=1098.959,170.811,433.566,177.335,16.339,152.015
C03230=1098.954,170.562,433.587,177.332,16.339,152.015
C03231=1098.948,170.313,433.609,177.328,16.339,152.016
C03232=1098.943,170.063,433.631,177.325,16.339,152.017
C03233=1098.937,169.815,433.653,177.322,16.340,152.017
C03234=1098.932,169.566,433.675,177.318,16.340,152.018
C03235=1098.926,169.317,433.697,177.315,16.340,152.019
C03236=1098.921,169.068,433.719,177.311,16.340,152.020
C03237=1098.914,168.819,433.741,177.309,16.340,152.020
C03238=1098.910,168.570,433.762,177.305,16.340,152.021
C03239=1098.903,168.321,433.785,177.302,16.340,152.022
C03240=1098.898,168.072,433.807,177.298,16.340,152.022
C03241=1098.892,167.823,433.828,177.295,16.341,152.023
C03242=1098.887,167.574,433.850,177.292,16.341,152.024
C03243=1098.881,167.325,433.872,177.288,16.341,152.025
C03244=1098.876,167.076,433.894,177.285,16.341,152.025
C03245=1098.870,166.827,433.915,177.282,16.341,152.026
C03246=1098.865,166.578,433.937,177.279,16.341,152.027
C03247=1098.859,166.329,433.959,177.275,16.341,152.027
C03248=1098.854,166.080,433.981,177.272,16.341,152.028
C03249=1098.848,165.831,434.002,177.269,16.342,152.029
C03250=1098.843,165.582,434.024,177.266,16.341,152.029
C03251=1098.837,165.333,434.046,177.262,16.341,152.030
C03252=1098.832,165.084,434.068,177.259,16.341,152.031
C03253=1098.826,164.835,434.089,177.256,16.342,152.031
C03254=1098.821,164.586,434.111,177.252,16.341,152.032
C03255=1098.815,164.337,434.133,177.249,16.341,152.033
C03256=1098.810,164.088,434.155,177.245,16.341,152.033
C03257=1098.804,163.839,434.176,177.243,16.342,152.034
C03258=1098.799,163.591,434.198,177.239,16.342,152.035
C03259=1098.793,163.341,434.220,177.236,16.342,152.035
C03260=1098.788,163.093,434.241,177.232,16.342,152.036
C03261=1098.782,162.843,434.263,177.230,16.342,152.037
C03262=1098.777,162.595,434.285,177.226,16.342,152.037
C03263=1098.771,162.346,434.306,177.223,16.342,152.038
C03264=1098.766,162.096,434.327,177.219,16.341,152.039
C03265=1098.760,161.847,434.349,177.217,16.342,152.039
C03266=1098.755,161.598,434.371,177.213,16.342,152.040
C03267=1098.749,161.349,434.392,177.210,16.342,152.041
C03268=1098.743,161.100,434.414,177.206,16.342,152.041
C03269=1098.738,160.852,434.435,177.204,16.342,152.042
C03270=1098.732,160.602,434.456,177.200,16.342,152.043
C03271=1098.726,160.328,434.480,177.196,16.342,152.044
C03272=1098.719,160.054,434.503,177.193,16.342,152.044
C03273=1098.713,159.780,434.527,177.189,16.342,152.045
C03274=1098.707,159.507,434.551,177.186,16.342,152.046
C03275=1098.701,159.257,434.572,177.182,16.342,152.047
C03276=1098.696,159.008,434.593,177.180,16.343,152.047
C03277=1098.690,158.759,434.615,177.176,16.343,152.048
C03278=1098.685,158.510,434.636,177.173,16.343,152.049
C03279=1098.679,158.260,434.657,177.169,16.342,152.049
C03280=1098.674,158.012,434.678,177.167,16.343,152.050
C03281=1098.667,157.763,434.700,177.163,16.343,152.051
C03282=1098.662,157.513,434.721,177.160,16.342,152.051
C03283=1098.657,157.265,434.742,177.157,16.343,152.052
C03284=1098.650,157.016,434.764,177.154,16.343,152.053
C03285=1098.646,156.766,434.785,177.150,16.343,152.053
C03286=1098.640,156.517,434.806,177.147,16.343,152.054
C03287=1098.634,156.269,434.828,177.144,16.343,152.054
C03288=1098.629,156.020,434.848,177.141,16.343,152.055
C03289=1098.623,155.770,434.870,177.137,16.343,152.056
C03290=1098.617,155.521,434.890,177.135,16.343,152.056
C03291=1098.612,155.273,434.912,177.131,16.343,152.057
C03292=1098.606,155.023,434.933,177.128,16.343,152.058
C03293=1098.600,154.774,434.954,177.124,16.343,152.058
C03294=1098.594,154.525,434.975,177.122,16.343,152.059
C03295=1098.589,154.276,434.996,177.118,16.343,152.060
C03296=1098.583,154.028,435.017,177.115,16.343,152.060
C03297=1098.578,153.778,435.038,177.112,16.343,152.061
C03298=1098.572,153.529,435.059,177.109,16.343,152.062
C03299=1098.567,153.280,435.080,177.105,16.343,152.062
C03300=1098.561,153.031,435.102,177.103,16.343,152.063
C03301=1098.555,152.782,435.122,177.099,16.343,152.064
C03302=1098.550,152.533,435.143,177.096,16.343,152.064
C03303=1098.544,152.283,435.164,177.093,16.343,152.065
C03304=1098.538,152.035,435.186,177.090,16.343,152.066
C03305=1098.533,151.786,435.206,177.087,16.343,152.066
C03306=1098.527,151.537,435.228,177.083,16.343,152.067
C03307=1098.522,151.287,435.248,177.081,16.343,152.067
C03308=1098.516,151.038,435.269,177.077,16.343,152.068
C03309=1098.510,150.789,435.291,177.074,16.343,152.069
C03310=1098.504,150.540,435.311,177.071,16.343,152.069
C03311=1098.499,150.292,435.332,177.068,16.343,152.070
C03312=1098.494,150.043,435.352,177.064,16.343,152.071
C03313=1098.488,149.793,435.373,177.061,16.343,152.071
C03314=1098.482,149.544,435.395,177.058,16.343,152.072
C03315=1098.477,149.295,435.415,177.055,16.343,152.073
C03316=1098.471,149.045,435.436,177.052,16.342,152.073
C03317=1098.465,148.797,435.457,177.049,16.343,152.074
C03318=1098.459,148.548,435.477,177.046,16.343,152.074
C03319=1098.454,148.299,435.498,177.042,16.342,152.075
C03320=1098.448,148.049,435.519,177.040,16.343,152.076
C03321=1098.443,147.801,435.540,177.036,16.342,152.076
C03322=1098.438,147.552,435.561,177.033,16.342,152.077
C03323=1098.432,147.303,435.581,177.030,16.343,152.078
C03324=1098.425,147.053,435.602,177.027,16.342,152.078
C03325=1098.420,146.804,435.623,177.023,16.342,152.079
C03326=1098.415,146.555,435.643,177.021,16.342,152.079
C03327=1098.409,146.306,435.663,177.017,16.342,152.080
C03328=1098.403,146.057,435.684,177.014,16.342,152.081
C03329=1098.397,145.808,435.705,177.011,16.342,152.081
C03330=1098.392,145.559,435.726,177.008,16.342,152.082
C03331=1098.386,145.310,435.746,177.005,16.342,152.083
C03332=1098.380,145.060,435.767,177.002,16.341,152.083
C03333=1098.375,144.811,435.787,176.999,16.342,152.084
C03334=1098.369,144.562,435.807,176.996,16.342,152.085
C03335=1098.363,144.288,435.830,176.992,16.342,152.085
C03336=1098.356,144.013,435.853,176.989,16.341,152.086
C03337=1098.351,143.739,435.876,176.985,16.341,152.087
C03338=1098.344,143.465,435.898,176.982,16.341,152.087
C03339=1098.339,143.216,435.919,176.979,16.342,152.088
C03340=1098.334,142.967,435.939,176.976,16.341,152.088
C03341=1098.327,142.717,435.959,176.973,16.341,152.089
C03342=1098.322,142.468,435.980,176.970,16.341,152.090
C03343=1098.317,142.219,436.001,176.967,16.341,152.090
C03344=1098.311,141.970,436.021,176.963,16.341,152.091
C03345=1098.305,141.722,436.042,176.961,16.341,152.091
C03346=1098.300,141.473,436.062,176.958,16.340,152.092
C03347=1098.294,141.224,436.082,176.954,16.340,152.093
C03348=1098.288,140.974,436.103,176.952,16.341,152.093
C03349=1098.283,140.724,436.123,176.948,16.340,152.094
C03350=1098.277,140.476,436.143,176.945,16.340,152.094
C03351=1098.272,140.226,436.164,176.943,16.340,152.095
C03352=1098.266,139.978,436.184,176.939,16.340,152.096
C03353=1098.261,139.729,436.204,176.936,16.339,152.096
C03354=1098.255,139.480,436.224,176.933,16.340,152.097
C03355=1098.249,139.231,436.245,176.930,16.339,152.097
C03356=1098.243,138.981,436.266,176.927,16.339,152.098
C03357=1098.237,138.732,436.285,176.924,16.339,152.099
C03358=1098.232,138.483,436.306,176.921,16.339,152.099
C03359=1098.226,138.234,436.326,176.918,16.338,152.100
C03360=1098.221,137.985,436.347,176.915,16.339,152.100
C03361=1098.215,137.736,436.366,176.912,16.339,152.101
C03362=1098.210,137.486,436.386,176.909,16.338,152.102
C03363=1098.204,137.238,436.406,176.906,16.339,152.102
C03364=1098.199,136.988,436.427,176.903,16.338,152.103
C03365=1098.193,136.740,436.447,176.900,16.338,152.103
C03366=1098.186,136.490,436.467,176.897,16.338,152.104
C03367=1098.181,136.240,436.487,176.894,16.338,152.104
C03368=1098.175,135.991,436.507,176.891,16.337,152.105
C03369=1098.170,135.742,436.527,176.888,16.337,152.106
C03370=1098.164,135.494,436.547,176.885,16.337,152.106
C03371=1098.159,135.244,436.568,176.882,16.337,152.107
C03372=1098.153,134.995,436.587,176.879,16.337,152.107
C03373=1098.147,134.746,436.607,176.876,16.337,152.108
C03374=1098.142,134.497,436.628,176.873,16.337,152.109
C03375=1098.136,134.248,436.648,176.870,16.337,152.109
C03376=1098.131,133.999,436.668,176.867,16.336,152.110
C03377=1098.125,133.750,436.687,176.864,16.336,152.110
C03378=1098.120,133.501,436.708,176.861,16.336,152.111
C03379=1098.114,133.251,436.727,176.858,16.336,152.111
C03380=1098.108,133.002,436.747,176.855,16.335,152.112
C03381=1098.103,132.753,436.768,176.852,16.335,152.112
C03382=1098.097,132.504,436.787,176.849,16.335,152.113
C03383=1098.091,132.255,436.807,176.846,16.335,152.113
C03384=1098.086,132.006,436.828,176.843,16.334,152.114
C03385=1098.080,131.756,436.847,176.840,16.334,152.115
C03386=1098.074,131.508,436.867,176.837,16.334,152.115
C03387=1098.068,131.258,436.886,176.834,16.334,152.116
C03388=1098.063,131.009,436.907,176.832,16.334,152.116
C03389=1098.057,130.760,436.927,176.828,16.334,152.117
C03390=1098.051,130.511,436.946,176.825,16.333,152.117
C03391=1098.045,130.262,436.966,176.823,16.333,152.118
C03392=1098.040,130.013,436.985,176.819,16.333,152.119
C03393=1098.034,129.763,437.006,176.816,16.333,152.119
C03394=1098.029,129.514,437.025,176.814,16.333,152.120
C03395=1098.023,129.265,437.045,176.810,16.332,152.120
C03396=1098.017,129.016,437.064,176.808,16.333,152.121
C03397=1098.011,128.767,437.084,176.805,16.332,152.121
C03398=1098.005,128.517,437.103,176.801,16.332,152.122
C03399=1097.999,128.244,437.125,176.798,16.331,152.123
C03400=1097.993,127.969,437.147,176.795,16.331,152.123
C03401=1097.987,127.694,437.169,176.792,16.331,152.124
C03402=1097.981,127.420,437.190,176.789,16.331,152.124
C03403=1097.975,127.171,437.210,176.786,16.330,152.125
C03404=1097.969,126.922,437.229,176.783,16.330,152.125
C03405=1097.963,126.673,437.249,176.780,16.330,152.126
C03406=1097.958,126.423,437.269,176.777,16.330,152.127
C03407=1097.952,126.174,437.288,176.774,16.330,152.127
C03408=1097.946,125.925,437.308,176.771,16.330,152.128
C03409=1097.941,125.675,437.328,176.768,16.329,152.128
C03410=1097.935,125.426,437.347,176.766,16.329,152.129
C03411=1097.929,125.177,437.367,176.762,16.329,152.129
C03412=1097.923,124.928,437.386,176.759,16.328,152.130
C03413=1097.918,124.680,437.406,176.757,16.328,152.130
C03414=1097.912,124.430,437.425,176.754,16.328,152.131
C03415=1097.907,124.181,437.444,176.751,16.328,152.131
C03416=1097.902,123.931,437.464,176.748,16.327,152.132
C03417=1097.896,123.682,437.484,176.745,16.327,152.133
C03418=1097.890,123.433,437.503,176.743,16.327,152.133
C03419=1097.884,123.183,437.522,176.739,16.326,152.134
C03420=1097.878,122.934,437.542,176.737,16.327,152.134
C03421=1097.873,122.686,437.561,176.734,16.326,152.135
C03422=1097.867,122.436,437.580,176.731,16.325,152.135
C03423=1097.862,122.187,437.600,176.728,16.326,152.136
C03424=1097.856,121.938,437.620,176.725,16.325,152.136
C03425=1097.850,121.689,437.639,176.722,16.324,152.137
C03426=1097.845,121.440,437.658,176.719,16.325,152.137
C03427=1097.839,121.190,437.677,176.716,16.324,152.138
C03428=1097.834,120.941,437.696,176.714,16.324,152.138
C03429=1097.828,120.692,437.716,176.711,16.324,152.139
C03430=1097.822,120.443,437.735,176.708,16.323,152.139
C03431=1097.817,120.194,437.754,176.705,16.323,152.140
C03432=1097.811,119.945,437.774,176.702,16.323,152.140
C03433=1097.805,119.695,437.793,176.700,16.322,152.141
C03434=1097.800,119.446,437.812,176.696,16.322,152.141
C03435=1097.794,119.196,437.831,176.694,16.321,152.142
C03436=1097.789,118.948,437.851,176.691,16.321,152.142
C03437=1097.783,118.699,437.870,176.688,16.320,152.143
C03438=1097.777,118.449,437.889,176.686,16.321,152.143
C03439=1097.772,118.200,437.909,176.682,16.320,152.144
C03440=1097.767,117.951,437.927,176.679,16.319,152.144
C03441=1097.761,117.702,437.947,176.677,16.320,152.145
C03442=1097.755,117.452,437.966,176.674,16.319,152.145
C03443=1097.749,117.203,437.985,176.671,16.319,152.146
C03444=1097.744,116.954,438.004,176.668,16.318,152.146
C03445=1097.739,116.705,438.023,176.665,16.318,152.147
C03446=1097.733,116.455,438.043,176.663,16.317,152.147
C03447=1097.728,116.206,438.061,176.660,16.317,152.148
C03448=1097.722,115.957,438.081,176.657,16.316,152.148
C03449=1097.717,115.708,438.100,176.655,16.316,152.149
C03450=1097.711,115.459,438.119,176.651,16.316,152.149
C03451=1097.706,115.209,438.138,176.649,16.315,152.150
C03452=1097.700,114.960,438.157,176.646,16.315,152.150
C03453=1097.694,114.712,438.176,176.643,16.314,152.151
C03454=1097.689,114.462,438.195,176.640,16.314,152.151
C03455=1097.683,114.213,438.214,176.637,16.314,152.152
C03456=1097.677,113.963,438.233,176.635,16.314,152.152
C03457=1097.672,113.714,438.251,176.632,16.313,152.153
C03458=1097.666,113.465,438.270,176.630,16.313,152.153
C03459=1097.660,113.215,438.289,176.627,16.312,152.154
C03460=1097.655,112.967,438.308,176.624,16.311,152.154
C03461=1097.650,112.717,438.327,176.621,16.312,152.155
C03462=1097.643,112.468,438.346,176.618,16.311,152.155
C03463=1097.638,112.194,438.367,176.615,16.310,152.156
C03464=1097.631,111.919,438.388,176.612,16.311,152.156
C03465=1097.625,111.644,438.408,176.609,16.310,152.157
C03466=1097.618,111.370,438.429,176.606,16.309,152.157
C03467=1097.613,111.121,438.448,176.603,16.309,152.158
C03468=1097.607,110.872,438.467,176.601,16.309,152.158
C03469=1097.602,110.622,438.485,176.598,16.308,152.159
C03470=1097.596,110.373,438.504,176.595,16.308,152.159
C03471=1097.590,110.124,438.523,176.592,16.307,152.160
C03472=1097.584,109.875,438.542,176.589,16.307,152.160
C03473=1097.580,109.625,438.560,176.587,16.307,152.161
C03474=1097.573,109.376,438.579,176.584,16.306,152.161
C03475=1097.567,109.127,438.598,176.581,16.306,152.161
C03476=1097.562,108.878,438.617,176.578,16.305,152.162
C03477=1097.556,108.628,438.635,176.575,16.304,152.162
C03478=1097.551,108.379,438.654,176.573,16.305,152.163
C03479=1097.545,108.130,438.673,176.570,16.304,152.163
C03480=1097.539,107.880,438.691,176.568,16.304,152.164
C03481=1097.534,107.632,438.710,176.565,16.303,152.164
C03482=1097.528,107.383,438.729,176.562,16.303,152.165
C03483=1097.522,107.132,438.747,176.559,16.302,152.165
C03484=1097.517,106.884,438.765,176.556,16.302,152.166
C03485=1097.511,106.635,438.785,176.554,16.302,152.166
C03486=1097.505,106.385,438.803,176.551,16.301,152.167
C03487=1097.500,106.136,438.821,176.549,16.300,152.167
C03488=1097.494,105.887,438.841,176.546,16.300,152.168
C03489=1097.488,105.638,438.858,176.543,16.300,152.168
C03490=1097.483,105.388,438.878,176.540,16.299,152.168
C03491=1097.477,105.139,438.895,176.538,16.299,152.169
C03492=1097.472,104.890,438.914,176.535,16.298,152.169
C03493=1097.465,104.641,438.933,176.532,16.298,152.170
C03494=1097.460,104.391,438.951,176.530,16.297,152.170
C03495=1097.454,104.142,438.970,176.527,16.296,152.171
C03496=1097.449,103.893,438.988,176.525,16.296,152.171
C03497=1097.443,103.644,439.007,176.521,16.296,152.172
C03498=1097.438,103.394,439.025,176.519,16.296,152.172
C03499=1097.432,103.145,439.043,176.516,16.295,152.172
C03500=1097.427,102.896,439.062,176.513,16.294,152.173
C03501=1097.421,102.646,439.081,176.511,16.294,152.173
C03502=1097.416,102.397,439.098,176.508,16.293,152.174
C03503=1097.410,102.148,439.118,176.506,16.293,152.174
C03504=1097.404,101.899,439.135,176.503,16.292,152.175
C03505=1097.399,101.649,439.154,176.500,16.292,152.175
C03506=1097.393,101.400,439.172,176.497,16.291,152.175
C03507=1097.387,101.151,439.190,176.495,16.291,152.176
C03508=1097.382,100.902,439.209,176.492,16.290,152.176
C03509=1097.376,100.652,439.227,176.489,16.289,152.177
C03510=1097.370,100.404,439.245,176.487,16.289,152.177
C03511=1097.365,100.154,439.264,176.484,16.289,152.178
C03512=1097.359,99.905,439.281,176.482,16.288,152.178
C03513=1097.353,99.656,439.300,176.479,16.288,152.179
C03514=1097.348,99.406,439.318,176.477,16.287,152.179
C03515=1097.342,99.157,439.336,176.474,16.287,152.179
C03516=1097.336,98.908,439.354,176.471,16.286,152.180
C03517=1097.331,98.658,439.373,176.468,16.285,152.180
C03518=1097.325,98.409,439.390,176.466,16.285,152.181
C03519=1097.319,98.160,439.409,176.463,16.285,152.181
C03520=1097.314,97.911,439.427,176.460,16.284,152.182
C03521=1097.308,97.661,439.445,176.458,16.284,152.182
C03522=1097.302,97.412,439.463,176.455,16.283,152.182
C03523=1097.297,97.162,439.482,176.453,16.283,152.183
C03524=1097.291,96.913,439.499,176.450,16.282,152.183
C03525=1097.285,96.664,439.518,176.447,16.282,152.184
C03526=1097.279,96.415,439.536,176.445,16.281,152.184
C03527=1097.273,96.141,439.555,176.442,16.280,152.185
C03528=1097.267,95.866,439.576,176.439,16.280,152.185
C03529=1097.261,95.592,439.596,176.436,16.279,152.186
C03530=1097.254,95.316,439.615,176.433,16.279,152.186
C03531=1097.249,95.068,439.633,176.430,16.278,152.186
C03532=1097.243,94.819,439.651,176.428,16.277,152.187
C03533=1097.238,94.569,439.669,176.425,16.277,152.187
C03534=1097.232,94.320,439.687,176.423,16.276,152.188
C03535=1097.226,94.070,439.705,176.420,16.276,152.188
C03536=1097.220,93.821,439.723,176.418,16.275,152.188
C03537=1097.215,93.572,439.741,176.415,16.274,152.189
C03538=1097.209,93.323,439.759,176.413,16.274,152.189
C03539=1097.204,93.074,439.777,176.410,16.273,152.190
C03540=1097.198,92.824,439.794,176.408,16.273,152.190
C03541=1097.192,92.575,439.812,176.405,16.272,152.190
C03542=1097.187,92.325,439.831,176.402,16.272,152.191
C03543=1097.181,92.076,439.849,176.399,16.271,152.191
C03544=1097.176,91.827,439.866,176.397,16.271,152.192
C03545=1097.170,91.578,439.884,176.394,16.270,152.192
C03546=1097.164,91.328,439.902,176.392,16.268,152.192
C03547=1097.159,91.079,439.920,176.389,16.268,152.193
C03548=1097.153,90.830,439.938,176.386,16.267,152.193
C03549=1097.147,90.580,439.956,176.384,16.267,152.194
C03550=1097.142,90.331,439.974,176.381,16.266,152.194
C03551=1097.136,90.082,439.991,176.379,16.266,152.194
C03552=1097.130,89.832,440.009,176.376,16.265,152.195
C03553=1097.125,89.583,440.027,176.374,16.265,152.195
C03554=1097.119,89.334,440.045,176.371,16.264,152.196
C03555=1097.113,89.085,440.062,176.369,16.264,152.196
C03556=1097.108,88.836,440.080,176.366,16.263,152.196
C03557=1097.101,88.586,440.098,176.364,16.262,152.197
C03558=1097.096,88.337,440.115,176.361,16.262,152.197
C03559=1097.090,88.088,440.133,176.359,16.261,152.198
C03560=1097.085,87.837,440.150,176.356,16.261,152.198
C03561=1097.079,87.588,440.168,176.354,16.260,152.198
C03562=1097.074,87.339,440.185,176.351,16.259,152.199
C03563=1097.067,87.090,440.203,176.349,16.259,152.199
C03564=1097.062,86.841,440.221,176.346,16.258,152.200
C03565=1097.056,86.592,440.238,176.344,16.258,152.200
C03566=1097.051,86.343,440.256,176.341,16.257,152.200
C03567=1097.045,86.093,440.274,176.339,16.256,152.201
C03568=1097.039,85.844,440.291,176.336,16.255,152.201
C03569=1097.034,85.595,440.309,176.334,16.255,152.201
C03570=1097.028,85.344,440.326,176.331,16.254,152.202
C03571=1097.022,85.095,440.344,176.329,16.254,152.202
C03572=1097.017,84.846,440.361,176.326,16.253,152.203
C03573=1097.011,84.597,440.379,176.324,16.253,152.203
C03574=1097.005,84.347,440.397,176.321,16.252,152.203
C03575=1097.000,84.098,440.413,176.319,16.251,152.204
C03576=1096.994,83.849,440.430,176.316,16.250,152.204
C03577=1096.988,83.600,440.448,176.314,16.250,152.204
C03578=1096.982,83.350,440.466,176.311,16.249,152.205
C03579=1096.977,83.101,440.484,176.309,16.248,152.205
C03580=1096.971,82.852,440.500,176.306,16.248,152.206
C03581=1096.966,82.603,440.518,176.304,16.247,152.206
C03582=1096.960,82.353,440.536,176.301,16.246,152.206
C03583=1096.954,82.103,440.553,176.299,16.246,152.207
C03584=1096.949,81.854,440.570,176.296,16.245,152.207
C03585=1096.943,81.605,440.588,176.294,16.244,152.207
C03586=1096.938,81.356,440.605,176.291,16.244,152.208
C03587=1096.931,81.106,440.622,176.289,16.243,152.208
C03588=1096.926,80.857,440.640,176.286,16.242,152.208
C03589=1096.920,80.608,440.657,176.284,16.242,152.209
C03590=1096.915,80.358,440.674,176.281,16.240,152.209
C03591=1096.909,80.084,440.694,176.278,16.240,152.210
C03592=1096.903,79.810,440.712,176.276,16.239,152.210
C03593=1096.896,79.535,440.731,176.273,16.238,152.210
C03594=1096.890,79.261,440.751,176.270,16.237,152.211
C03595=1096.885,79.011,440.768,176.268,16.237,152.211
C03596=1096.879,78.762,440.785,176.265,16.236,152.211
C03597=1096.873,78.512,440.802,176.263,16.236,152.212
C03598=1096.868,78.263,440.820,176.260,16.235,152.212
C03599=1096.862,78.014,440.837,176.258,16.234,152.212
C03600=1096.856,77.765,440.853,176.255,16.233,152.213
C03601=1096.851,77.516,440.871,176.253,16.233,152.213
C03602=1096.845,77.266,440.888,176.250,16.232,152.214
C03603=1096.839,77.016,440.906,176.249,16.231,152.214
C03604=1096.833,76.767,440.922,176.246,16.230,152.214
C03605=1096.828,76.518,440.940,176.243,16.230,152.215
C03606=1096.823,76.268,440.956,176.241,16.229,152.215
C03607=1096.816,76.019,440.973,176.239,16.228,152.215
C03608=1096.811,75.770,440.990,176.236,16.227,152.216
C03609=1096.805,75.520,441.008,176.234,16.227,152.216
C03610=1096.799,75.271,441.024,176.231,16.226,152.216
C03611=1096.794,75.022,441.042,176.229,16.225,152.217
C03612=1096.788,74.772,441.059,176.226,16.224,152.217
C03613=1096.782,74.523,441.076,176.224,16.224,152.217
C03614=1096.777,74.274,441.093,176.221,16.223,152.218
C03615=1096.771,74.025,441.110,176.219,16.222,152.218
C03616=1096.765,73.775,441.126,176.216,16.221,152.218
C03617=1096.759,73.526,441.144,176.214,16.221,152.219
C03618=1096.753,73.276,441.161,176.212,16.220,152.219
C03619=1096.748,73.026,441.177,176.209,16.219,152.219
C03620=1096.743,72.777,441.195,176.207,16.219,152.220
C03621=1096.737,72.528,441.211,176.204,16.218,152.220
C03622=1096.732,72.278,441.228,176.203,16.217,152.220
C03623=1096.726,72.029,441.246,176.200,16.216,152.221
C03624=1096.720,71.780,441.262,176.198,16.216,152.221
